# B&R Automation Studio project Panasonic_LinkaPowerCP2_A2021055 (part 6)

#### TP_Unlock.st
```iecst
(********************************************************************
 * COPYRIGHT -- Bernecker + Rainer
 ********************************************************************
 * Library: RFID
 * File: TP_Unlock.st
 * Author: houx
 * Created: March 25, 2009
*****************************************************************
;FuB: 			TP_Unlock
;*****************************************************************
Discription:
	This FuB is used to open a password-protected transponder so that all register can be edited.
	transponder key 4102 can not be used with this FuB.
	The password, protection word,and control word can only be modified after a valid TP_Unlock.
Parameter:
	Input:
		Enable(BOOL)	: The function block is only executed when enable is <> 0
	Output:
		Error(BOOL)		: Error = 0 (No Error) Error = 1(see ErrorID)
		ErrorID(UDINT)	: Number and Description in Error Table
		Busy(BOOL)		: Fub working on
		Ident(UDINT)	: Interface ID
		Done(BOOL)		: success, if TRUE
Author:	Xiaoguang Hou
		B&R Eggelsberg
;
;History:	V1.00.0 - 02 Sep 2008 : first create
				V3.00.0 - 25 Mar 2009 : update for serial interface transponder and created under AS3.0

 ********************************************************************
 * Implementation of library RFID
 ********************************************************************)

FUNCTION_BLOCK TP_Unlock

IF	(Enable	=	1)	THEN
	IF ((Done = 0) AND (Error = 0)) THEN
		Busy:=TRUE;
		IF TypeOK = FALSE THEN
			CASE StepType OF
(*	------------------------------------------------	open the interface, get the internal Ident	----------------------------------------------------*)
				OPEN:
					FrameXOpenStruct(enable := 1,device := Ident);
					status.XOPEN 			:= FrameXOpenStruct.status;
					IF (status.XOPEN = 0) THEN
						StepType            := WRITE ;
					ELSE
						StepType            := OPEN ;
						Error               := TRUE;
						ErrorID             := status.XOPEN;
						Busy                := 0;
					END_IF
				WRITE:
				memset(ADR(WriteData),0,SIZEOF(WriteData));
				strcpy(ADR(WriteData),ADR('tag,0,0,#crc$R$L'));
				FrameGetBufferStruct(enable:= 1, ident:= FrameXOpenStruct.ident);
				sendbuffer				:= FrameGetBufferStruct.buffer;
				sendbufferlength		:= FrameGetBufferStruct.buflng;
				status.GetBuffer		:= FrameGetBufferStruct.status;
				IF	(status.GetBuffer = 0)	THEN
					memcpy(sendbuffer,ADR(WriteData),sendbufferlength);
					FrameWriteStruct(enable := 1, ident := FrameXOpenStruct.ident, buffer := sendbuffer,buflng :=strlen(ADR(WriteData)));
					status.WRITE 				:=	FrameWriteStruct.status;
					StepType              		:=	READ;
				    IF (status.WRITE <> 0) THEN
						FrameReleaseOutputBufferStruct(enable:=1,ident:=FrameXOpenStruct.ident,buffer:=sendbuffer,buflng:=strlen(ADR(WriteData)));
						status.RoBuffer			:= FrameReleaseOutputBufferStruct.status;
						IF	(status.RoBuffer <> 0)	THEN
							ErrorID   	:= status.RoBuffer;
						END_IF
						FrameReleaseOutputBufferStruct.enable := 0;
						FrameWriteStruct.enable 	:=	0;
						FrameGetBufferStruct.enable	:=	0;
					END_IF
				ELSE
					ErrorID 	:= status.GetBuffer;
					Error   	:= 1;
					Busy    	:= 0;
					StepType	:= OPEN;
					TypeOK		:= FALSE;
					FrameGetBufferStruct.enable	:= 0;
				END_IF

				READ:
					FrameReadStruct(enable:=1,ident:=FrameXOpenStruct.ident);
					ReadBuffer       	:=	FrameReadStruct.buffer;
					ReadBufferLength	:=	FrameReadStruct.buflng;
					status.READ      	:=	FrameReadStruct.status;
					IF  (status.READ = 0) THEN
						memset(ADR(ReadData),0,SIZEOF(ReadData));
						memcpy(ADR(ReadData),ReadBuffer,ReadBufferLength);                   (* copy read data into read buffer *)
						FrameReadStruct.enable	:= 0;
				        FrameReleaseBufferStruct(enable:=1, ident:=FrameXOpenStruct.ident, buffer:=ReadBuffer,buflng:=ReadBufferLength);        (* release read buffer *)
				        status.ReleaseBuffer	:=FrameReleaseBufferStruct.status;
				        IF (status.ReleaseBuffer=0) THEN
					        FrameReleaseBufferStruct.enable:=0;
							AN[0]	:= ReadData[0];
							AN[1]	:= ReadData[1];
							AN[2]	:= ReadData[2];
							IF (memcmp(ADR(AN),ADR('ack'),3) = 0) THEN
								IF (memcmp(ADR(ReadData),ADR('ack,0,4150'),10) = 0) THEN
									StepType	:=	OPEN;
									TypeOK		:=	TRUE;
								ELSE
									StepType	:= 	OPEN;
									ErrorID		:=	rfidError_unlock_wrongType;          (*  hier ein Error difinieren soll  *)
									Error   	:=	1;
									Busy    	:=	0;
									TypeOK		:=	FALSE;
								END_IF
							ELSE
								StepType	:= 	OPEN;
								ErrorID		:=	rfidError_unlock_failed;          (*  hier ein Error difinieren soll  *)
								Error   	:=	1;
								Busy    	:=	0;
								TypeOK		:=	FALSE;
							END_IF
						ELSE
							StepType	:=	OPEN;
							Error     	:=	1;
							ErrorID   	:=	status.ReleaseBuffer;
							Busy      	:=	0;
							TypeOK		:=	FALSE;
						END_IF
					ELSE
						memset(ADR(ReadData),0,SIZEOF(ReadData));
					END_IF
			END_CASE
		END_IF
		IF	(TypeOK	= TRUE)	THEN
			string1	:=	'li,0,';
			string2	:=	',#crc$R$L';
			CMD		:=	strcat(ADR(string1),Data);
			CMD		:=	strcat(ADR(string1),ADR(string2));
			memset(ADR(WriteData),0,SIZEOF(WriteData));
			strcpy(ADR(WriteData),ADR(string1));
			CASE StepWrite OF
				OPEN:
					FrameXOpenStruct(enable := 1,device := Ident);
					status.XOPEN 			:= FrameXOpenStruct.status;
					IF (status.XOPEN = 0) THEN
						StepWrite            := WRITE ;
					ELSE
						StepWrite            := OPEN ;
						Error               := TRUE;
						ErrorID             := status.XOPEN;
						Busy                := 0;
					END_IF
				WRITE:
					FrameGetBufferStruct(enable:= 1, ident:= FrameXOpenStruct.ident);
					sendbuffer					:= FrameGetBufferStruct.buffer;
					sendbufferlength		:= FrameGetBufferStruct.buflng;
					status.GetBuffer		:= FrameGetBufferStruct.status;
					IF	(status.GetBuffer = 0)	THEN
						memcpy(sendbuffer,ADR(WriteData),sendbufferlength);
						FrameWriteStruct(enable := 1, ident := FrameXOpenStruct.ident, buffer := sendbuffer,buflng := strlen(ADR(WriteData)));
						status.WRITE 				:=	FrameWriteStruct.status;
					    IF (status.WRITE = FALSE) THEN
					    	StepWrite              		:=	READ;
							FrameWriteStruct.enable 	:=	0;
							FrameGetBufferStruct.enable	:=	0;
						ELSE
							ErrorID 				:= status.WRITE;
							Error   				:= 1;
							Busy    				:= 0;
							StepWrite				:= OPEN;
							TypeOK					:= FALSE;
							FrameWriteStruct.enable := 0;
							FrameGetBufferStruct.enable	:= 0;
							FrameReleaseOutputBufferStruct(enable:=1,ident:=FrameXOpenStruct.ident,buffer:=sendbuffer,buflng:= sendbufferlength);
							status.RoBuffer			:= FrameReleaseOutputBufferStruct.status;
							IF	(status.RoBuffer <> 0)	THEN
								StepWrite 	:= OPEN;
								Error     	:= TRUE;
								ErrorID   	:= status.RoBuffer;
								Busy      	:= 0;
								TypeOK		:= FALSE;
								FrameReleaseOutputBufferStruct.enable := 0;
							END_IF
						END_IF
					ELSE
						ErrorID 	:= status.GetBuffer;
						Error   	:= 1;
						Busy    	:= 0;
						StepWrite	:= OPEN;
						TypeOK		:= FALSE;
						FrameGetBufferStruct.enable	:= 0;
					END_IF
			    READ:
				    FrameReadStruct(enable := 1,ident:=FrameXOpenStruct.ident);
					ReadBuffer			:=	FrameReadStruct.buffer;
					ReadBufferLength	:=	FrameReadStruct.buflng;
					status.READ			:=	FrameReadStruct.status;
					IF  (status.READ = 0)  THEN
						memset(ADR(ReadData),0,SIZEOF(ReadData));
						memcpy(ADR(ReadData),ReadBuffer,ReadBufferLength);
						FrameReadStruct.enable := 0;
				        FrameReleaseBufferStruct(enable:=1, ident:=FrameXOpenStruct.ident, buffer:=ReadBuffer,buflng:=ReadBufferLength);
				        status.ReleaseBuffer	:=	FrameReleaseBufferStruct.status;
				        IF status.ReleaseBuffer=0 THEN
							FrameReleaseBufferStruct.enable:=0;
							AN[0]	:= ReadData[0];
							AN[1]	:= ReadData[1];
							AN[2]	:= ReadData[2];
							IF (memcmp(ADR(AN),ADR('ack'),3)) = 0 THEN
								StepWrite		:=	WRITE;
							 	Busy			:=	0;
							 	Done			:=	1;
								TypeOK			:=	FALSE;
							ELSIF	(memcmp(ADR(AN),ADR('nak'),3)) = 0 THEN
								ERROR[0]	:=	ReadData[6];
								ERROR[1]	:=	ReadData[7];
								ERROR[2]	:=	ReadData[8];
								Error		:=	1;
								ErrorID		:=	atoi(ADR(ERROR)) ;
								Busy		:=	0;
								TypeOK		:=	FALSE;
								StepWrite	:=	WRITE;
							ELSE
								Error			:=	1;
								ErrorID			:=	rfidError_unlock_failed ;(* unknow answer *)
								Busy			:=	0;
								TypeOK			:=	FALSE;
								StepWrite		:=	WRITE;
							END_IF
						ELSE
							Error			:=	1;
							ErrorID			:=	status.ReleaseBuffer ;
							Busy			:=	0;
							TypeOK			:=	FALSE;
							StepWrite		:=	WRITE;
					    END_IF
					ELSE
						memset(ADR(ReadData),0,SIZEOF(ReadData));
					END_IF
			END_CASE
		END_IF
	END_IF
ELSE
	Busy	:=	0;
	Error	:=	0;
	ErrorID	:=	0;
	Done	:=	0;
END_IF
END_FUNCTION_BLOCK
```

#### TP_Lock.st
```iecst
(********************************************************************
 * COPYRIGHT -- Bernecker + Rainer
 ********************************************************************
 * Library: RFID
 * File: TP_Lock.st
 * Author: houx
 * Created: March 25, 2009
 *****************************************************************
;FuB: 			TP_Lock
;*****************************************************************
Discription:
	If a password-protected transponder was opened with the TP_Unlock, it can be locked again with this FuB
	From this point on, password-protected areas can no longer be edited.
	if the transponder is removed from the reading range of the transponder reader, then it is locked automatically.
Parameter:
	Input:
		Enable(BOOL)	: The function block is only executed when enable is <> 0
	Output:
		Error(BOOL)		: Error = 0 (No Error) Error = 1(see ErrorID)
		ErrorID(UDINT)	: Number and Description in Error Table
		Busy(BOOL)		: Fub working on
		Ident(UDINT)	: Interface ID
		Done(BOOL)		: success, if TRUE
;Author:	Xiaoguang Hou
;			B&R Eggelsberg
;
;History:	V1.00.0 - 02 Sep 2008 : first create
				V3.00.0 - 25 Mar 2009 : update for serial interface transponder and created under AS3.0
;
;******************************************************************

 ********************************************************************
 * Implementation of library RFID
 ********************************************************************)
(*TODO: Add your comment here*)
FUNCTION_BLOCK TP_Lock

IF Enable = TRUE THEN
	IF ((Done = 0) AND (Error = 0)) THEN
		Busy:=TRUE;
		IF TypeOK = FALSE THEN
			CASE StepType OF
(*	------------------------------------------------	open the interface, get the internal Ident	----------------------------------------------------*)
				OPEN:
					FrameXOpenStruct(enable := 1,device := Ident);
					status.XOPEN 			:= FrameXOpenStruct.status;
					IF (status.XOPEN = 0) THEN
						StepType            := WRITE ;
					ELSE
						StepType            := OPEN ;
						Error               := TRUE;
						ErrorID             := status.XOPEN;
						Busy                := 0;
					END_IF
				WRITE:
					memset(ADR(WriteData),0,SIZEOF(WriteData));
					strcpy(ADR(WriteData),ADR('tag,0,0,#crc$R$L'));
					FrameGetBufferStruct(enable:= 1, ident:= FrameXOpenStruct.ident);
					sendbuffer				:= FrameGetBufferStruct.buffer;
					sendbufferlength		:= FrameGetBufferStruct.buflng;
					status.GetBuffer		:= FrameGetBufferStruct.status;
					IF	(status.GetBuffer = 0)	THEN
						memcpy(sendbuffer,ADR(WriteData),sendbufferlength);
						FrameWriteStruct(enable := 1, ident := FrameXOpenStruct.ident, buffer := sendbuffer,buflng := strlen(ADR(WriteData)));
						status.WRITE 				:=	FrameWriteStruct.status;
					    StepType              		:=	READ;
					    IF (status.WRITE <> 0) THEN
							FrameReleaseOutputBufferStruct(enable:=1,ident:=FrameXOpenStruct.ident,buffer:=sendbuffer,buflng:= strlen(ADR(WriteData)));
							status.RoBuffer			:= FrameReleaseOutputBufferStruct.status;
							IF	(status.RoBuffer <> 0)	THEN
								ErrorID   	:= status.RoBuffer;
							END_IF
						END_IF
						FrameWriteStruct.enable := 0;
						FrameGetBufferStruct.enable	:= 0;
						FrameReleaseOutputBufferStruct.enable := 0;
					ELSE
						ErrorID 	:= status.GetBuffer;
						Error   	:= 1;
						Busy    	:= 0;
						StepType	:= OPEN;
						TypeOK		:= FALSE;
						FrameGetBufferStruct.enable	:= 0;
					END_IF
				READ:
					FrameReadStruct(enable:=1,ident:=FrameXOpenStruct.ident);
					ReadBuffer       	:=	FrameReadStruct.buffer;
					ReadBufferLength	:=	FrameReadStruct.buflng;
					status.READ      	:=	FrameReadStruct.status;
					IF  (status.READ = 0) THEN
						memset(ADR(ReadData),0,SIZEOF(ReadData));
						memcpy(ADR(ReadData),ReadBuffer,ReadBufferLength);                   (* copy read data into read buffer *)
						FrameReadStruct.enable	:= 0;
				        FrameReleaseBufferStruct(enable:=1, ident:=FrameXOpenStruct.ident, buffer:=ReadBuffer,buflng:=ReadBufferLength);        (* release read buffer *)
				        status.ReleaseBuffer	:=FrameReleaseBufferStruct.status;
				        IF (status.ReleaseBuffer=0) THEN
					        FrameReleaseBufferStruct.enable:=0;
							AN[0]	:= ReadData[0];
							AN[1]	:= ReadData[1];
							AN[2]	:= ReadData[2];
							IF (memcmp(ADR(AN),ADR('ack'),3) = 0) THEN
								IF (memcmp(ADR(ReadData),ADR('ack,0,4150,#02d0$R$L'),SIZEOF('ack,0,4150,#02d0$R$L')) = 0) THEN
									StepType	:=	OPEN;
									TypeOK		:=	TRUE;
									StepLOCK	:=	WRITE;
								ELSE
									StepType	:= 	OPEN;
									ErrorID		:=	rfidError_lock_wrongType;          (*  hier ein Error difinieren soll  *)
									Error   	:=	1;
									Busy    	:=	0;
									TypeOK		:=	FALSE;
								END_IF
							ELSE
								StepType	:= 	OPEN;
								ErrorID		:=	rfidError_lock_failed;          (*  hier ein Error difinieren soll  *)
								Error   	:=	1;
								Busy    	:=	0;
								TypeOK		:=	FALSE;
							END_IF
						ELSE
							StepType	:=	OPEN;
							Error     	:=	1;
							ErrorID   	:=	status.ReleaseBuffer;
							Busy      	:=	0;
							TypeOK		:=	FALSE;
						END_IF
					ELSE
						memset(ADR(ReadData),0,SIZEOF(ReadData));
					END_IF
			END_CASE
		END_IF
		IF TypeOK = TRUE THEN
			CASE StepLOCK OF
				WRITE:
					memset(ADR(WriteData),0,SIZEOF(WriteData));
					strcpy(ADR(WriteData),ADR('re,0,#crc$R$L'));
					FrameGetBufferStruct(enable:= 1, ident:= FrameXOpenStruct.ident);
					sendbuffer				:= FrameGetBufferStruct.buffer;
					sendbufferlength		:= FrameGetBufferStruct.buflng;
					status.GetBuffer		:= FrameGetBufferStruct.status;
					IF	(status.GetBuffer = 0)	THEN
						memcpy(sendbuffer,ADR(WriteData),sendbufferlength);
						FrameWriteStruct(enable := 1, ident := FrameXOpenStruct.ident, buffer := sendbuffer,buflng := strlen(ADR(WriteData)));
						status.WRITE 				:=	FrameWriteStruct.status;
					   	StepLOCK              		:=	READ;
					    IF (status.WRITE <> 0) THEN
							FrameReleaseOutputBufferStruct(enable:=1,ident:=FrameXOpenStruct.ident,buffer:=sendbuffer,buflng:= sendbufferlength);
							status.RoBuffer			:= FrameReleaseOutputBufferStruct.status;
							IF	(status.RoBuffer <> 0)	THEN
								ErrorID   	:= status.RoBuffer;
							END_IF
						END_IF
						FrameWriteStruct.enable := 0;
						FrameGetBufferStruct.enable	:= 0;
						FrameReleaseOutputBufferStruct.enable := 0;
					ELSE
						ErrorID 	:= status.GetBuffer;
						Error   	:= 1;
						Busy    	:= 0;
						StepLOCK	:= WRITE;
						TypeOK		:= FALSE;
						FrameGetBufferStruct.enable	:= 0;
					END_IF
				READ:
				    FrameReadStruct(enable := 1,ident:=FrameXOpenStruct.ident);
					ReadBuffer			:= FrameReadStruct.buffer;
					ReadBufferLength	:= FrameReadStruct.buflng;
					status.READ			:= FrameReadStruct.status;
					IF  (status.READ = 0) THEN
						memset(ADR(ReadData),0,SIZEOF(ReadData));
						memcpy(ADR(ReadData),ReadBuffer,ReadBufferLength);                   (* copy read data into read buffer *)
						FrameReadStruct.enable 	:= 0;
				        FrameReleaseBufferStruct(enable:=1, ident:=FrameXOpenStruct.ident, buffer:=ReadBuffer,buflng:=ReadBufferLength);        (* release read buffer *)
				        status.ReleaseBuffer	:= FrameReleaseBufferStruct.status;
				        IF (status.ReleaseBuffer=0) THEN
						    FrameReleaseBufferStruct.enable	:= 0;
							AN[0]	:= ReadData[0];
							AN[1]	:= ReadData[1];
							AN[2]	:= ReadData[2];
							IF (memcmp(ADR(AN),ADR('ack'),3)) = 0 THEN
								StepLOCK  := WRITE;
								Done      := 1;
								Busy      := 0;
								TypeOK	  := FALSE;
							ELSIF	(memcmp(ADR(AN),ADR('nak'),3)) = 0 THEN
								ERROR[0]	:=	ReadData[6];
								ERROR[1]	:=	ReadData[7];
								ERROR[2]	:=	ReadData[8];
								Error		:=	1;
								ErrorID		:=	atoi(ADR(ERROR)) ;
								Busy		:=	0;
								TypeOK		:=	FALSE;
								StepLOCK	:=	WRITE;
							ELSE
								StepLOCK  := WRITE;
								Error     := 1;
								ErrorID   := rfidError_lock_failed; (* unknow answer *)
								Busy      := 0;
								TypeOK	  := FALSE;
							END_IF
						ELSE
							StepLOCK  := WRITE;
							Error     := 1;
							ErrorID   := status.ReleaseBuffer;
							Busy      := 0;
							TypeOK	  := FALSE;
					    END_IF
					ELSE
						memset(ADR(ReadData),0,SIZEOF(ReadData));
					END_IF
			END_CASE
		END_IF
	END_IF
ELSE
	Busy 	:= 0;
	ErrorID := 0;
	Error 	:= 0;
	Done 	:= 0;
END_IF
END_FUNCTION_BLOCK
```

#### TP_PWProtect.st
```iecst
(********************************************************************
 * COPYRIGHT -- Bernecker + Rainer
 ********************************************************************
 * Library: RFID
 * File: TP_PWProtect.st
 * Author: houx
 * Created: March 25, 2009
 *****************************************************************
;FuB: 			TP_PWProtect
;*****************************************************************
Discription:
	This FuB is used to write the password
	before a new password can be written, a valid TP_Unlock must be done.
Parameter:
	Input:
		Enable(BOOL)	:The function block is only executed when enable is <> 0
		Data(UDINT)		:Pointer to Password. whick should be write in transponder.
	Output:
		Error(BOOL)		:Error = 0 (No Error) Error = 1(see ErrorID)
		ErrorID(UDINT)	:Number and Description in Error Table
		Busy(BOOL)		:Fub working on
		Done			:success, if TRUE
;Author:	Xiaoguang Hou
;			B&R Eggelsberg
;
;History: 	V1.00.0 - 02 Sep 2008 first create
				V3.00.0 - 25 Mar 2009  update for serial interface transponder reader and created under AS3.0
;
;******************************************************************

 ********************************************************************
 * Implementation of library RFID
 ********************************************************************)

(*TODO: Add your comment here*)
FUNCTION_BLOCK TP_PWProtect

IF	(Enable	=	1)	THEN
	IF ((Done = 0) AND (Error = 0)) THEN
		Busy:=TRUE;
		IF TypeOK = FALSE THEN
			CASE StepType OF
(*	------------------------------------------------	open the interface, get the internal Ident	----------------------------------------------------*)
				OPEN:
					FrameXOpenStruct(enable := 1,device := Ident);
					status.XOPEN 			:= FrameXOpenStruct.status;
					IF (status.XOPEN = 0) THEN
						StepType            := WRITE ;
					ELSE
						StepType            := OPEN ;
						Error               := TRUE;
						ErrorID             := status.XOPEN;
						Busy                := 0;
					END_IF
				WRITE:
					memset(ADR(WriteData),0,SIZEOF(WriteData));
					strcpy(ADR(WriteData),ADR('tag,0,0,#crc$R$L'));
					FrameGetBufferStruct(enable:= 1, ident:= FrameXOpenStruct.ident);
					sendbuffer				:= FrameGetBufferStruct.buffer;
					sendbufferlength		:= FrameGetBufferStruct.buflng;
					status.GetBuffer		:= FrameGetBufferStruct.status;
					IF	(status.GetBuffer = 0)	THEN
						memcpy(sendbuffer,ADR(WriteData),sendbufferlength);
						FrameWriteStruct(enable := 1, ident := FrameXOpenStruct.ident, buffer := sendbuffer,buflng := strlen(ADR(WriteData)));
						status.WRITE 				:=	FrameWriteStruct.status;
					    StepType              		:=	READ;
					    IF (status.WRITE <> 0) THEN
							FrameReleaseOutputBufferStruct(enable:=1,ident:=FrameXOpenStruct.ident,buffer:=sendbuffer,buflng:= strlen(ADR(WriteData)));
							status.RoBuffer			:= FrameReleaseOutputBufferStruct.status;
							IF	(status.RoBuffer <> 0)	THEN
								ErrorID	:=	status.RoBuffer;
							END_IF
						END_IF
						FrameWriteStruct.enable := 0;
						FrameGetBufferStruct.enable	:= 0;
						FrameReleaseOutputBufferStruct.enable := 0;
					ELSE
						ErrorID 	:= status.GetBuffer;
						Error   	:= 1;
						Busy    	:= 0;
						StepType	:= OPEN;
						TypeOK		:= FALSE;
						FrameGetBufferStruct.enable	:= 0;
					END_IF

				READ:
					FrameReadStruct(enable:=1,ident:=FrameXOpenStruct.ident);
					ReadBuffer       	:=	FrameReadStruct.buffer;
					ReadBufferLength	:=	FrameReadStruct.buflng;
					status.READ      	:=	FrameReadStruct.status;
					IF  (status.READ = 0) THEN
						memset(ADR(ReadData),0,SIZEOF(ReadData));
						memcpy(ADR(ReadData),ReadBuffer,ReadBufferLength);                   (* copy read data into read buffer *)
						FrameReadStruct.enable	:= 0;
				        FrameReleaseBufferStruct(enable:=1, ident:=FrameXOpenStruct.ident, buffer:=ReadBuffer,buflng:=ReadBufferLength);        (* release read buffer *)
				        status.ReleaseBuffer	:=FrameReleaseBufferStruct.status;
				        IF (status.ReleaseBuffer=0) THEN
					        FrameReleaseBufferStruct.enable:=0;
							IF (memcmp(ADR(ReadData),ADR('ack,0,4150,#02d0$R$L'),SIZEOF('ack,0,4150,#02d0$R$L')) = 0) THEN
								StepType	:=	OPEN;
								TypeOK		:=	TRUE;
								StepWrite	:=	WRITE;
							ELSE
								StepType	:= 	OPEN;
								ErrorID		:=	rfidError_password_wrongType;         (*   hier ein Error difinieren soll  *)
								Error   	:=	1;
								Busy    	:=	0;
								TypeOK		:=	FALSE;
							END_IF
						ELSE
							StepType	:=	OPEN;
							Error     	:=	1;
							ErrorID   	:=	status.ReleaseBuffer;
							Busy      	:=	0;
							TypeOK		:=	FALSE;
						END_IF
					ELSE
						memset(ADR(ReadData),0,SIZEOF(ReadData));
					END_IF
			END_CASE
		END_IF
		IF	(TypeOK	= TRUE)	THEN
			string1	:=	'wp,0,';
			string2	:=	',#crc$R$L';
			CMD		:=	strcat(ADR(string1),Data);
			CMD		:=	strcat(ADR(string1),ADR(string2));
			memset(ADR(WriteData),0,SIZEOF(WriteData));
			memcpy(ADR(WriteData),ADR(string1),SIZEOF(string1));
			CASE StepWrite OF
				WRITE:
					FrameGetBufferStruct(enable:= 1, ident:= FrameXOpenStruct.ident);
					sendbuffer				:= FrameGetBufferStruct.buffer;
					sendbufferlength		:= FrameGetBufferStruct.buflng;
					status.GetBuffer		:= FrameGetBufferStruct.status;
					IF	(status.GetBuffer = 0)	THEN
						memcpy(sendbuffer,ADR(WriteData),sendbufferlength);
						FrameWriteStruct(enable := 1, ident := FrameXOpenStruct.ident, buffer := sendbuffer,buflng := strlen(ADR(WriteData)));
						status.WRITE 				:=	FrameWriteStruct.status;
					    StepWrite              		:=	READ;
					    IF (status.WRITE <> 0) THEN
							FrameReleaseOutputBufferStruct(enable:=1,ident:=FrameXOpenStruct.ident,buffer:=sendbuffer,buflng:=strlen(ADR(WriteData)) );
							status.RoBuffer			:= FrameReleaseOutputBufferStruct.status;
							IF	(status.RoBuffer <> 0)	THEN
								ErrorID	:=	status.RoBuffer;
							END_IF
						END_IF
						FrameWriteStruct.enable := 0;
						FrameGetBufferStruct.enable	:= 0;
						FrameReleaseOutputBufferStruct.enable := 0;
					ELSE
						ErrorID 	:= status.GetBuffer;
						Error   	:= 1;
						Busy    	:= 0;
						StepWrite	:= WRITE;
						TypeOK		:= FALSE;
						FrameGetBufferStruct.enable	:= 0;
					END_IF

			    READ:
				    FrameReadStruct(enable := 1,ident:=FrameXOpenStruct.ident);
					ReadBuffer			:=	FrameReadStruct.buffer;
					ReadBufferLength	:=	FrameReadStruct.buflng;
					status.READ			:=	FrameReadStruct.status;
					IF  (status.READ = 0)  THEN
						memset(ADR(ReadData),0,SIZEOF(ReadData));
						memcpy(ADR(ReadData),ReadBuffer,ReadBufferLength);
						FrameReadStruct.enable := 0;
				        FrameReleaseBufferStruct(enable:=1, ident:=FrameXOpenStruct.ident, buffer:=ReadBuffer,buflng:=ReadBufferLength);
				        status.ReleaseBuffer	:=	FrameReleaseBufferStruct.status;
				        IF status.ReleaseBuffer=0 THEN
							FrameReleaseBufferStruct.enable:=0;
							memset(ADR(AN),0,SIZEOF(AN));
							AN[0]	:= ReadData[0];
							AN[1]	:= ReadData[1];
							AN[2]	:= ReadData[2];
							IF (memcmp(ADR(AN),ADR('ack'),3)) = 0 THEN
								StepWrite		:=	WRITE;
							 	Busy			:=	0;
							 	Done			:=	1;
								TypeOK			:=	FALSE;
							ELSIF	(memcmp(ADR(AN),ADR('nak'),3)) = 0 THEN
								ERROR[0]	:=	ReadData[6];
								ERROR[1]	:=	ReadData[7];
								ERROR[2]	:=	ReadData[8];
								Error			:=	1;
								ErrorID			:=	atoi(ADR(ERROR)) ;
								Busy			:=	0;
								TypeOK			:=	FALSE;
								StepWrite		:=	WRITE;
							ELSE
								Error			:=	1;
								ErrorID			:=	rfidError_password_failed ;
								Busy			:=	0;
								TypeOK			:=	FALSE;
								StepWrite		:=	WRITE;
							END_IF
						ELSE
							Error			:=	1;
							ErrorID			:=	status.ReleaseBuffer ;
							Busy			:=	0;
							TypeOK			:=	FALSE;
							StepWrite		:=	WRITE;
					    END_IF
					ELSE
						memset(ADR(ReadData),0,SIZEOF(ReadData));
					END_IF
			END_CASE
		END_IF
	END_IF
ELSE
	Busy	:=	0;
	Error	:=	0;
	ErrorID	:=	0;
	Done	:=	0;
END_IF
END_FUNCTION_BLOCK
```

#### TP_OnOff.st
```iecst
(********************************************************************
 * COPYRIGHT -- Bernecker + Rainer
 ********************************************************************
 * Library: RFID
 * File: TP_OnOff.st
 * Author: houx
 * Created: March 25, 2009
 *****************************************************************
;FuB: 			TP_OnOff
;*****************************************************************
Discription:
	This FuB turn the 125 kHz carrier frequency of the Transponder reader/writer On/Off.
	This Fub can work without any Transponder in the range of Reader.
	Standard Configuration is frequency on.
	Be aware that no Transponder key can be read if frequency is turned off.
Parameter:
	Input:
		Enable(BOOL)	:	The function block is only executed when enable is <> 0
		Ident(UDINT)	:	Interface Ident from TP_Init.
   		Mode(BOOL)		:	frequency On:Mode=TRUE, frequency Off: Mode:=FALSE;
	Output:
		Error(BOOL)		:	Error = 0 (No Error) Error = 1(see ErrorID)
		ErrorID(UDINT)	:	Number and Description in Error Table
		Busy(BOOL)		:	if TRUE , Fub working on.
		Done(BOOL) 		:	if TRUE, success
Author:	Xiaoguang Hou
		B&R Eggelsberg

History: 	V1.00.0 - 02 Sep 2008 first create
				V3.00.0 - 25 Mar 2009  update for serial interface transponder reader and created under AS3.0

;******************************************************************

 ********************************************************************
 * Implementation of library RFID
 ********************************************************************)

(*TODO: Add your comment here*)
FUNCTION_BLOCK TP_OnOff

(*------------------------------------	Start	--------------------------------*)
IF Enable=1 THEN
	IF ((Done = 0) AND (Error = 0)) THEN
		Busy:=TRUE;
		CASE StepOnOff OF
(*	------------------------------------------------	open the interface, get the internal Ident	----------------------------------------------------*)
			OPEN:
				FrameXOpenStruct(enable := TRUE,device := Ident);
				status.XOPEN 			:= FrameXOpenStruct.status;
				IF (status.XOPEN = 0) THEN
					StepOnOff               := WRITE ;
					FrameXOpenStruct.enable:=FALSE;
				ELSE
					StepOnOff               := OPEN ;
					Error                   := TRUE;
					ErrorID                 := status.XOPEN;
					Busy                    := FALSE;
				END_IF

			WRITE:						(*------	write RF Command to	Reader	---------*)
				IF (Mode = TRUE) THEN
					memset(ADR(WriteData),0,SIZEOF(WriteData));
					strcpy(ADR(WriteData),ADR('rf,0,1,#crc$R$L'));
				ELSIF	(Mode = FALSE)	THEN
					memset(ADR(WriteData),0,SIZEOF(WriteData));
					strcpy(ADR(WriteData),ADR('rf,0,0,#crc$R$L'));
				END_IF
				(*------	get sendbuffer	---------*)
				FrameGetBufferStruct(enable:= TRUE, ident:= FrameXOpenStruct.ident);
				sendbuffer				:= FrameGetBufferStruct.buffer;
				sendbufferlength		:= FrameGetBufferStruct.buflng;
				status.GetBuffer		:= FrameGetBufferStruct.status;
				IF	(status.GetBuffer = 0)	THEN							 (*------	no error	---------*)
					memcpy(sendbuffer,ADR(WriteData),sendbufferlength);
					FrameWriteStruct(enable := TRUE, ident := FrameXOpenStruct.ident, buffer := sendbuffer,buflng :=strlen(ADR(WriteData)) );
					status.WRITE 				:=	FrameWriteStruct.status;
			        IF (status.WRITE <> 0) THEN
						FrameReleaseOutputBufferStruct(enable:=TRUE,ident:=FrameXOpenStruct.ident,buffer:=sendbuffer,buflng:= strlen(ADR(WriteData)));
						status.RoBuffer			:= FrameReleaseOutputBufferStruct.status;
						IF	(status.RoBuffer <> 0)	THEN
							ErrorID	:=	status.RoBuffer;
						END_IF
					ELSE
			        	StepOnOff              		:=	READ;
						FrameWriteStruct.enable := FALSE;
						FrameGetBufferStruct.enable	:= FALSE;
						FrameReleaseOutputBufferStruct.enable := FALSE;
					END_IF
				(*------	if get sendbuffer error	---------*)
				ELSE
					ErrorID 	:= status.GetBuffer;
					Error   	:= TRUE;
					Busy    	:= FALSE;
					StepOnOff	:= OPEN;
					FrameGetBufferStruct.enable	:= FALSE;
				END_IF

	    	READ:						(*	read out the feedback	*)
			    FrameReadStruct(enable := 1,ident:=FrameXOpenStruct.ident);
				ReadBuffer				:=FrameReadStruct.buffer;
				ReadBufferLength		:=FrameReadStruct.buflng;
				status.READ				:=FrameReadStruct.status;
				IF  (status.READ = 0) THEN
					memset(ADR(ReadData),0,SIZEOF(ReadData));
					memcpy(ADR(ReadData),ReadBuffer,ReadBufferLength);	(*	copy the answer	out in ReadData	*)
					FrameReadStruct.enable := 0;
			        FrameReleaseBufferStruct(enable:=1, ident:=FrameXOpenStruct.ident, buffer:=ReadBuffer,buflng:=ReadBufferLength);	(*	release the buffer	*)
			        status.ReleaseBuffer   := FrameReleaseBufferStruct.status;
			        IF (status.ReleaseBuffer=0) THEN
			        	FrameReleaseBufferStruct.enable	:= 0;
			        	AN[0]	:= ReadData[0];
						AN[1]	:= ReadData[1];
						AN[2]	:= ReadData[2];
						IF (memcmp(ADR(AN),ADR('ack'),3) = 0) THEN				(*--- positiv answer ----*)
							StepOnOff   := CLOSE;
						ELSE
							StepOnOff   := OPEN;								(*	negativ answer or unknow answer	*)
							Error     	:= 1;
							ErrorID   	:= rfidError_rf_failed;
							Busy      	:= 0;
						END_IF
					ELSE														(*	if buffer release error	*)
							StepOnOff   := OPEN;
							Error     	:= 1;
							ErrorID   	:= status.ReleaseBuffer;
							Busy     	:= 0;
			        END_IF
				ELSE
					memset(ADR(ReadData),0,SIZEOF(ReadData));
				END_IF
			CLOSE:
				FRM_close_0(enable :=1 , ident :=FrameXOpenStruct.ident);
				IF FRM_close_0.status=FALSE THEN
					Done      	:= 1;
					Busy      	:= 0;
					StepOnOff:=OPEN;
				END_IF
		END_CASE
	END_IF
ELSE                                          (*------- if enable = False ,then all output variable back to zero -------*)
	Error:=0;
	ErrorID:=0;
	Busy:=0;
	Done:=0;
END_IF
END_FUNCTION_BLOCK
```

#### TP_Crc.st
```iecst
(********************************************************************
 * COPYRIGHT -- Bernecker + Rainer
 ********************************************************************
 * Library: RFID
 * File: TP_Crc.st
 * Author: houx
 * Created: March 25, 2009
*****************************************************************
;FuB: 			TP_CRC
;*****************************************************************
Discription:
	This FuB can specify whether the transponder reader should check the checksum wenn a command string is received.
	This Fub can work without any Transponder in the range of Reader.
Parameter:
	Input: 	Enable(BOOL)	: The function block is only executed when enable is <> 0.
			Ident(UDINT)	: Interface Ident.
			Mode(BOOL)		: checksum On:Mode=TRUE, checksum Off: Mode:=FALSE;
	Output: Error(BOOL)		: Error = 0 (No Error) Error = 1(see ErrorID).
			ErrorID(UDINT)	: Number and description in error table.
			Busy(BOOL)		: FuB is working on.
			Done(BOOL)		: if TRUE, success.
Author:	Xiaoguang Hou
		B&R Eggelsberg

History: 	V1.00.0 - 02 Sep 2008 first create
				V3.00.0 - 25 Mar 2009  update for serial interface transponder readerand created under AS3.0
;
;******************************************************************

 ********************************************************************
 * Implementation of library RFID
 ********************************************************************)

(*TODO: Add your comment here*)
FUNCTION_BLOCK TP_Crc

IF Enable=1 THEN
	IF ((Done = 0) AND (Error = 0)) THEN
		Busy:=TRUE;
		CASE StepCRC OF
(*	------------------------------------------------	open the interface, get the internal Ident	----------------------------------------------------*)
			OPEN:
				FrameXOpenStruct(enable := 1,device := Ident);
				status.XOPEN 			:= FrameXOpenStruct.status;
				IF (status.XOPEN = 0) THEN
					StepCRC             := WRITE ;
					FrameXOpenStruct.enable:=FALSE;
				ELSE
					StepCRC             := OPEN ;
					Error               := TRUE;
					ErrorID             := status.XOPEN;
					Busy                := 0;
				END_IF
			WRITE:
				IF 	(Mode = TRUE) THEN
					memset(ADR(WriteData),0,SIZEOF(WriteData));
					strcpy(ADR(WriteData),ADR('cc,0,1,#01ce$R$L'));
				ELSIF (Mode = FALSE) THEN
					memset(ADR(WriteData),0,SIZEOF(WriteData));
					strcpy(ADR(WriteData),ADR('cc,0,0,#01cd$R$L'));
				END_IF
				FrameGetBufferStruct(enable:= 1, ident:= FrameXOpenStruct.ident);
				sendbuffer				:= FrameGetBufferStruct.buffer;
				sendbufferlength		:= FrameGetBufferStruct.buflng;
				status.GetBuffer		:= FrameGetBufferStruct.status;
				IF	(status.GetBuffer = 0)	THEN
					memcpy(sendbuffer,ADR(WriteData),sendbufferlength);
					FrameWriteStruct(enable := 1, ident := FrameXOpenStruct.ident, buffer := sendbuffer, buflng := strlen(ADR(WriteData)));
					status.WRITE 				:=	FrameWriteStruct.status;

			    	IF (status.WRITE <> 0) THEN
						FrameReleaseOutputBufferStruct(enable:=1,ident:=FrameXOpenStruct.ident,buffer:=sendbuffer,buflng:= strlen(ADR(WriteData)));
						status.RoBuffer			:= FrameReleaseOutputBufferStruct.status;
						IF	(status.RoBuffer <> 0)	THEN
							ErrorID:=status.RoBuffer;
						END_IF
					ELSE
			   			FrameWriteStruct.enable := 0;
						FrameGetBufferStruct.enable	:= 0;
						FrameReleaseOutputBufferStruct.enable := 0;
						StepCRC					:= READ;
					END_IF
				ELSE
					ErrorID 	:= status.GetBuffer;
					Error   	:= 1;
					Busy    	:= 0;
					StepCRC		:= OPEN;
					FrameGetBufferStruct.enable	:= 0;
				END_IF

		    READ:
			    FrameReadStruct(enable := 1,ident:=FrameXOpenStruct.ident);
				ReadBuffer			:= FrameReadStruct.buffer;
				ReadBufferLength	:= FrameReadStruct.buflng;
				status.READ			:= FrameReadStruct.status;
				IF  (status.READ = 0) THEN
					memset(ADR(ReadData),0,SIZEOF(ReadData));
					memcpy(ADR(ReadData),ReadBuffer,ReadBufferLength);                   (* copy read data into read buffer *)
					FrameReadStruct.enable 	:= 0;
			        FrameReleaseBufferStruct(enable:=1, ident:=FrameXOpenStruct.ident, buffer:=ReadBuffer,buflng:=ReadBufferLength);        (* release read buffer *)
			        status.ReleaseBuffer	:= FrameReleaseBufferStruct.status;
			        IF (status.ReleaseBuffer=0) THEN
				        FrameReleaseBufferStruct.enable	:=0;
		        		AN[0]	:= ReadData[0];
						AN[1]	:= ReadData[1];
						AN[2]	:= ReadData[2];
						IF (memcmp(ADR(AN),ADR('ack'),3) = 0) THEN
							StepCRC   := CLOSE;
						ELSE
							StepCRC   := OPEN;
							Error     := 1;
							ErrorID   := rfidError_crc_failed; (*	negativ answer *)
							Busy      := 0;
						END_IF
					ELSE
							StepCRC   := OPEN;
							Error     := 1;
							ErrorID   := status.ReleaseBuffer;
							Busy      := 0;
			        END_IF
				ELSE
					memset(ADR(ReadData),0,SIZEOF(ReadData));
				END_IF
			CLOSE:
				FRM_close_0(enable :=1 , ident :=FrameXOpenStruct.ident);
				IF FRM_close_0.status=FALSE  THEN
					Done      := 1;
					Busy      := 0;
					StepCRC   := OPEN;
				END_IF
		END_CASE
	END_IF
ELSE
	Error   := 0;
	ErrorID := 0;
	Busy    := 0;
	Done    := 0;
END_IF

END_FUNCTION_BLOCK
```

#### TP_Write.st
```iecst
(********************************************************************
 * COPYRIGHT -- Bernecker + Rainer
 ********************************************************************
 * Library: RFID
 * File: TP_Write.st
 * Author: houx
 * Created: March 25, 2009
 ****************************************************************
;FuB: 			TP_Write
;*****************************************************************
Discription:
	This FuB is used to write the registers of the transponder.
	for this to work, the transponder must not be password-protected or a valid TP_unlock must be carried out beforehand.
	Be aware that Register 1 and 2 of TP 4150 are used for the control and protectionwords.
	Only modify these registers,if you are familiar with their Function. In addition, avalid login is needed.
Parameter:
	Input:
		Enable(BOOL)	: The function block is only executed when enable is <> 0
		RegNr(USINT)	: Number of the register, which should be write in
		Data(UDINT)		: pointer to input Data
	Output:
		Error(BOOL)		: Error = 0 (No Error) Error = 1(see ErrorID)
		ErrorID(UDINT)	: Number and Description in Error Table
		Busy(BOOL)		: Fub working on
		Ident(UDINT)	: Interface ID
		Done(BOOL)		:success, if TRUE
Author:	Xiaoguang Hou
		B&R Eggelsberg
;
History: 	V1.00.0 - 02 Sep 2008 first create
				V3.00.0 - 25 Mar 2009  update for serial interface transponder reader and created under AS3.0
;
 ********************************************************************
 * Implementation of library RFID
 ********************************************************************)

(*TODO: Add your comment here*)
FUNCTION_BLOCK TP_Write

IF (Enable = 1) THEN
	IF ((Done = 0) AND (Error = 0)) THEN
		Busy:=TRUE;
		IF TypeOK = FALSE THEN
			CASE StepType OF
(*	------------------------------------------------	open the interface, get the internal Ident	----------------------------------------------------*)
				OPEN:
					FrameXOpenStruct(enable := 1,device := Ident);
					status.XOPEN 			:= FrameXOpenStruct.status;
					IF (status.XOPEN = 0) THEN
						StepType            := WRITE ;
					ELSE
						StepType            := OPEN ;
						Error               := TRUE;
						ErrorID             := status.XOPEN;
						Busy                := 0;
					END_IF
				WRITE:
					memset(ADR(WriteData),0,SIZEOF(WriteData));
					strcpy(ADR(WriteData),ADR('tag,0,0,#crc$R$L'));
					FrameGetBufferStruct(enable:= 1, ident:= FrameXOpenStruct.ident);
					sendbuffer				:= FrameGetBufferStruct.buffer;
					sendbufferlength		:= FrameGetBufferStruct.buflng;
					status.GetBuffer		:= FrameGetBufferStruct.status;
					IF	(status.GetBuffer = 0)	THEN
						memcpy(sendbuffer,ADR(WriteData),sendbufferlength);
						FrameWriteStruct(enable := 1, ident := FrameXOpenStruct.ident, buffer := sendbuffer,buflng := strlen(ADR(WriteData)));
						status.WRITE 				:=	FrameWriteStruct.status;
						StepType				:= READ;
					    IF (status.WRITE <> 0) THEN
							FrameReleaseOutputBufferStruct(enable:=1,ident:=FrameXOpenStruct.ident,buffer:=sendbuffer,buflng:= strlen(ADR(WriteData)));
							status.RoBuffer			:= FrameReleaseOutputBufferStruct.status;
							IF	(status.RoBuffer <> 0)	THEN
								ErrorID	:=	status.RoBuffer;
							END_IF
						END_IF
						FrameWriteStruct.enable := 0;
						FrameGetBufferStruct.enable	:= 0;
						FrameReleaseOutputBufferStruct.enable := 0;
					ELSE
						ErrorID 	:= status.GetBuffer;
						Error   	:= 1;
						Busy    	:= 0;
						StepType	:= OPEN;
						TypeOK		:= FALSE;
						FrameGetBufferStruct.enable	:= 0;
					END_IF

				READ:
					FrameReadStruct(enable:=1,ident:=FrameXOpenStruct.ident);
					ReadBuffer       	:=	FrameReadStruct.buffer;
					ReadBufferLength	:=	FrameReadStruct.buflng;
					status.READ      	:=	FrameReadStruct.status;
					IF  (status.READ = 0) THEN
						memset(ADR(ReadData),0,SIZEOF(ReadData));
						memcpy(ADR(ReadData),ReadBuffer,ReadBufferLength);                   (* copy read data into read buffer *)
						FrameReadStruct.enable	:= 0;
				        FrameReleaseBufferStruct(enable:=1, ident:=FrameXOpenStruct.ident, buffer:=ReadBuffer,buflng:=ReadBufferLength);        (* release read buffer *)
				        status.ReleaseBuffer	:=FrameReleaseBufferStruct.status;
				        IF (status.ReleaseBuffer=0) THEN
					        FrameReleaseBufferStruct.enable:=0;
							AN[0]		 :=	ReadData[0];
							AN[1]		 := ReadData[1];
							AN[2]		 := ReadData[2];
							IF	(memcmp(ADR(AN),ADR('ack'),3) = 0)	THEN
								memset(ADR(KeyType),0,SIZEOF(KeyType));
								KeyType[0] 	 :=	ReadData[6];
								KeyType[1] 	 := ReadData[7];
								KeyType[2] 	 := ReadData[8];
								KeyType[3] 	 := ReadData[9];
								IF (memcmp(ADR(KeyType),ADR('4150'),4) = 0) THEN
									StepType	:=	OPEN;
									TypeOK		:=	TRUE;
								ELSIF	(memcmp(ADR(KeyType),ADR('4102'),4) = 0) THEN
									StepType	:= 	OPEN;
									ErrorID		:=	rfidError_write_wrongType;         (*   wrong Type *)
									Error   	:=	1;
									Busy    	:=	0;
									TypeOK		:=	FALSE;
								ELSE
									StepType		:= 	OPEN;
									ErrorID			:=	rfidError_write_wrongType;            (* unknow type to write  *)
									Error   		:=	1;
									Busy    		:=	0;
									TypeOK			:=	FALSE;
								END_IF
							ELSIF	(memcmp(ADR(AN),ADR('nak'),3) = 0)	THEN
								StepType		:=	OPEN;
								ErrorID			:=	rfidError_write_failed; (* negativ answer *)
								Error   		:=	1;
								Busy    		:=	0;
								TypeOK			:=	FALSE;
							ELSE
								StepType	:= 	OPEN;
								ErrorID		:=	rfidError_write_failed; (* unknow answer *)
								Error   	:=	1;
								Busy    	:=	0;
								TypeOK			:=	FALSE;
							END_IF
						ELSE
							StepType	:=	OPEN;
							Error     	:=	1;
							ErrorID   	:=	status.ReleaseBuffer;
							Busy      	:=	0;
							TypeOK		:=	FALSE;
						END_IF
					ELSE
						memset(ADR(ReadData),0,SIZEOF(ReadData));
					END_IF
			END_CASE
		END_IF
		IF	(TypeOK	= TRUE)	THEN
			IF	(CommandReady = 0) THEN
				IF	(RegNr > 31) THEN
					Error	:=	1;
					ErrorID	:=	rfidError_write_wrongRegNr; (* hier soll ein Fehler Meldung difiniert werden: password Register, please use TP_Password Fub*)
					Busy	:=	0;
					TypeOK	:=	FALSE;
				ELSE
					itoa(RegNr,ADR(string1));
					string2:='wr,0,';
					string3:=',#crc$R$L';
					CMD	:=	strcat(ADR(string2),ADR(string1));
					CMD	:=	strcat(ADR(string2),ADR(','));
					CMD	:=	strcat(ADR(string2),Data);
					CMD	:=	strcat(ADR(string2),ADR(string3));
					memset(ADR(WriteData),0,SIZEOF(WriteData));
					strcpy(ADR(WriteData),ADR(string2));
					CommandReady:=	1;
					StepWrite	:=	WRITE;
				END_IF
			ELSE
				CASE StepWrite OF
					WRITE:
						FrameGetBufferStruct(enable:= 1, ident:= FrameXOpenStruct.ident);
						sendbuffer				:= FrameGetBufferStruct.buffer;
						sendbufferlength		:= FrameGetBufferStruct.buflng;
						status.GetBuffer		:= FrameGetBufferStruct.status;
						IF	(status.GetBuffer = 0)	THEN
							memcpy(sendbuffer,ADR(WriteData),sendbufferlength);
							FrameWriteStruct(enable := 1, ident := FrameXOpenStruct.ident, buffer := sendbuffer,buflng := strlen(ADR(WriteData)));
							status.WRITE 				:=	FrameWriteStruct.status;
						    StepWrite              		:=	READ;
						    IF (status.WRITE <> 0) THEN
								FrameReleaseOutputBufferStruct(enable:=1,ident:=FrameXOpenStruct.ident,buffer:=sendbuffer,buflng:= strlen(ADR(WriteData)));
								status.RoBuffer			:= FrameReleaseOutputBufferStruct.status;
								IF	(status.RoBuffer <> 0)	THEN
									ErrorID	:=	status.RoBuffer;
								END_IF
							END_IF
							FrameWriteStruct.enable := 0;
							FrameGetBufferStruct.enable	:= 0;
							FrameReleaseOutputBufferStruct.enable := 0;
						ELSE
							ErrorID 		:= status.GetBuffer;
							Error   		:= 1;
							Busy    		:= 0;
							StepWrite		:= WRITE;
							TypeOK			:= FALSE;
							CommandReady	:=	0;
							FrameGetBufferStruct.enable	:= 0;
						END_IF

			    	READ:
				    	FrameReadStruct(enable := 1,ident:=FrameXOpenStruct.ident);
						ReadBuffer			:=	FrameReadStruct.buffer;
						ReadBufferLength	:=	FrameReadStruct.buflng;
						status.READ			:=	FrameReadStruct.status;
						IF  (status.READ = 0)  THEN
							memset(ADR(ReadData),0,SIZEOF(ReadData));
							memcpy(ADR(ReadData),ReadBuffer,ReadBufferLength);
							FrameReadStruct.enable := 0;
					        FrameReleaseBufferStruct(enable:=1, ident:=FrameXOpenStruct.ident, buffer:=ReadBuffer,buflng:=ReadBufferLength);
					        status.ReleaseBuffer	:=	FrameReleaseBufferStruct.status;
					        IF status.ReleaseBuffer=0 THEN
								FrameReleaseBufferStruct.enable:=0;
					        	AN[0]	:= ReadData[0];
								AN[1]	:= ReadData[1];
								AN[2]	:= ReadData[2];
								IF (memcmp(ADR(AN),ADR('ack'),3) = 0) THEN
									StepWrite		:=	WRITE;
								 	Busy			:=	0;
								 	Done			:=	1;
									CommandReady	:=	0;
									TypeOK			:=	FALSE;
								ELSIF	(memcmp(ADR(AN),ADR('nak'),3) = 0)	THEN
									ERROR[0]	:=	ReadData[6];
									ERROR[1]	:=	ReadData[7];
									ERROR[2]	:=	ReadData[8];
									Error			:=	1;
									ErrorID			:=	rfidError_write_failed ;
									Busy			:=	0;
									CommandReady	:=	0;
									TypeOK			:=	FALSE;
									StepWrite		:=	WRITE;
								ELSE
									Error			:=	1;
									ErrorID			:=	rfidError_write_failed;
									Busy			:=	0;
									CommandReady	:=	0;
									TypeOK			:=	FALSE;
									StepWrite		:=	WRITE;
								END_IF
							ELSE
								Error			:=	1;
								ErrorID			:=	status.ReleaseBuffer ;
								Busy			:=	0;
								CommandReady	:=	0;
								TypeOK			:=	FALSE;
								StepWrite		:=	WRITE;
					       	END_IF
						ELSE
							memset(ADR(ReadData),0,SIZEOF(ReadData));
						END_IF
				END_CASE
			END_IF
		END_IF
	END_IF
ELSE
	Busy	:= 0;
	Error   := 0;
	ErrorID := 0;
	Done	:= 0;
END_IF
END_FUNCTION_BLOCK
```

#### TP_Read.st
```iecst
(********************************************************************
 * COPYRIGHT -- Bernecker + Rainer
 ********************************************************************
 * Library: RFID
 * File: TP_Read.st
 * Author: houx
 * Created: March 25, 2009
 *****************************************************************
;FuB: 			TP_Read
;*****************************************************************
Discription:
	This FuB is used to read the registers of the transponder.
	for this to work, the transponder must not be password-protected or a valid TP_unlock needs to be performed beforehand.
Parameter:
	Input:
		Enable(BOOL)	: The function block is only executed when enable is <> 0
		RegNr(USINT)	: Number of the register, which should be read out
	Output:
		Error(BOOL)		: Error = 0 (No Error) Error = 1(see ErrorID)
		ErrorID(BOOL)	: Number and Description in Error Table
		Busy(BOOL)		: Fub working on
		Data(BOOL)		: pointer to output Data.
		Done(BOOL)		: success, if TRUE
Author:	Xiaoguang Hou
		B&R Eggelsberg

History: 	V1.00.0 - 02 Sep 2008 first create
				V3.00.0 - 25 Mar 2009  update for serial interface transponder reader and created under AS3.0

 ********************************************************************
 * Implementation of library RFID
 ********************************************************************)

(*TODO: Add your comment here*)
FUNCTION_BLOCK TP_Read

    IF Enable = TRUE THEN
        IF ((Done = 0) AND (Error = 0)) THEN
            Busy:=TRUE;
            IF (TypeOK = FALSE) THEN
                CASE StepType OF
                    (*	------------------------------------------------	open the interface, get the internal Ident	----------------------------------------------------*)
                    OPEN:
                        FrameXOpenStruct.mode:=ADR(' /RIT=200 ');			(* long receive idle time for receive the data*)
                        FrameXOpenStruct(enable := 1,device := Ident);
                        status.XOPEN 			:= FrameXOpenStruct.status;
                        IF (status.XOPEN = 0) THEN
                            StepType            := WRITE ;
                            FrameXOpenStruct.enable := 0;
                        ELSE
                            StepType            := OPEN ;
                            Error               := TRUE;
                            ErrorID             := status.XOPEN;
                            Busy                := 0;
                            FrameXOpenStruct.enable := 0;
                        END_IF
                    WRITE:
                        memset(ADR(WriteData),0,SIZEOF(WriteData));
                        strcpy(ADR(WriteData),ADR('tag,0,#crc$R$L'));
                        FrameGetBufferStruct(enable:= 1, ident:= FrameXOpenStruct.ident);
                        sendbuffer					:= FrameGetBufferStruct.buffer;
                        sendbufferlength		:= FrameGetBufferStruct.buflng;
                        status.GetBuffer		:= FrameGetBufferStruct.status;
                        IF	(status.GetBuffer = 0)	THEN
                            memcpy(sendbuffer,ADR(WriteData),sendbufferlength);
                            FrameWriteStruct(enable := 1, ident := FrameXOpenStruct.ident, buffer := sendbuffer,buflng := strlen(ADR(WriteData)) );
                            status.WRITE 				:=	FrameWriteStruct.status;
                            IF (status.WRITE <> 0) THEN
                                FrameReleaseOutputBufferStruct(enable:=1,ident:=FrameXOpenStruct.ident,buffer:=sendbuffer,buflng:= strlen(ADR(WriteData)));
                                status.RoBuffer				:= FrameReleaseOutputBufferStruct.status;
                                IF (status.RoBuffer <> 0) THEN
                                    ErrorID:=status.RoBuffer;
                                END_IF
                            ELSE
                                StepType	:=	READ;
                                FrameWriteStruct.enable 	:= 0;
                                FrameGetBufferStruct.enable	:= 0;
                                FrameReleaseOutputBufferStruct.enable := 0;
                            END_IF
                        ELSE
                            ErrorID 	:= status.GetBuffer;
                            Error   	:= 1;
                            Busy    	:= 0;
                            StepType	:= OPEN;
                            TypeOK		:= FALSE;
                            FrameGetBufferStruct.enable	:= 0;
                        END_IF
                    READ:
                        FrameReadStruct(enable:=1,ident:=FrameXOpenStruct.ident);
                        ReadBuffer       	:=	FrameReadStruct.buffer;
                        ReadBufferLength	:=	FrameReadStruct.buflng;
                        status.READ      	:=	FrameReadStruct.status;
                        IF  (status.READ = 0) THEN
                            memset(ADR(ReadData),0,SIZEOF(ReadData));
                            memcpy(ADR(ReadData),ReadBuffer,ReadBufferLength);                   (* copy read data into read buffer *)
                            FrameReadStruct.enable	:= 0;
                            FrameReleaseBufferStruct(enable:=1, ident:=FrameXOpenStruct.ident, buffer:=ReadBuffer,buflng:=ReadBufferLength);        (* release read buffer *)
                            status.ReleaseBuffer	:=FrameReleaseBufferStruct.status;
                            IF (status.ReleaseBuffer=0) THEN
                                FrameReleaseBufferStruct.enable:=0;
                                AN[0]		 := ReadData[0];
                                AN[1]		 := ReadData[1];
                                AN[2]		 := ReadData[2];
                                IF	(memcmp(ADR(AN),ADR('ack'),3) = 0)	THEN
                                    memset(ADR(KeyType),0,SIZEOF(KeyType));
                                    KeyType[0] 	 := ReadData[6];
                                    KeyType[1] 	 := ReadData[7];
                                    KeyType[2] 	 := ReadData[8];
                                    KeyType[3] 	 := ReadData[9];
                                    IF (memcmp(ADR(KeyType),ADR('4150'),4) = 0) THEN
                                        StepType		:=	OPEN;
                                        Done         	:=	FALSE;
                                        Busy         	:=	0;
                                        CommandReady	:=	0;
                                        TypeOK			:=	TRUE;
                                    ELSIF	(memcmp(ADR(KeyType),ADR('4102'),4) = 0) THEN
                                        memset(ADR(data),0,SIZEOF(data));
                                        data[0] 	 	:=	ReadData[11];
                                        data[1] 	 	:=	ReadData[12];
                                        data[2] 	 	:=	ReadData[13];
                                        data[3] 	 	:=	ReadData[14];
                                        data[4] 	 	:=	ReadData[15];
                                        data[5] 	 	:=	ReadData[16];
                                        data[6] 	 	:=	ReadData[17];
                                        data[7] 	 	:=	ReadData[18];
                                        data[8] 	 	:=	ReadData[19];
                                        data[9] 	 	:=	ReadData[20];
                                        Data			:=	ADR(data);
                                        StepType		:=	OPEN;
                                        Done         	:=	1;
                                        Busy         	:=	0;
                                        CommandReady	:=	0;
                                        TypeOK			:=	FALSE;
                                    ELSE
                                        StepType		:= 	OPEN;
                                        ErrorID			:=	rfidError_read_wrongType;            (* wrong type to read  *)
                                        Error   		:=	1;
                                        Busy    		:=	0;
                                        CommandReady	:=	0;
                                        TypeOK			:=	FALSE;
                                    END_IF
                                ELSIF	(memcmp(ADR(AN),ADR('nak'),3) = 0)	THEN
                                    StepType		:= 	OPEN;
                                    ErrorID			:=	rfidError_read_failed; (* negativ answer *)
                                    Error   		:=	1;
                                    Busy    		:=	0;
                                    CommandReady	:=	0;
                                    TypeOK			:=	FALSE;
                                ELSE
                                    StepType		:=	OPEN;
                                    ErrorID			:=	rfidError_read_failed; (* unknow answer *)
                                    Error   		:=	1;
                                    Busy    		:=	0;
                                    CommandReady	:=	0;
                                    TypeOK			:=	FALSE;
                                END_IF
                            ELSE
                                StepType		:=	OPEN;
                                Error     		:=	1;
                                ErrorID   		:=	status.ReleaseBuffer;
                                Busy      		:=	0;
                                CommandReady	:=	0;
                                TypeOK			:=	FALSE;
                            END_IF
                        ELSE
                            memset(ADR(ReadData),0,SIZEOF(ReadData));
                        END_IF
                END_CASE
            END_IF
            IF	(TypeOK = TRUE) THEN
                IF CommandReady = 0 THEN
                    IF  ((0 < RegNr) AND (RegNr <34)) THEN
                        memset(ADR(WriteData),0,SIZEOF(WriteData));
                        CASE RegNr OF
                            REG1:
                                strcpy(ADR(WriteData),ADR('rdm,0,1,1,#crc$R$L'));
                            REG2:
                                strcpy(ADR(WriteData),ADR('rdm,0,2,1,#crc$R$L'));
                            REG3:
                                strcpy(ADR(WriteData),ADR('rdm,0,3,1,#crc$R$L'));
                            REG4:
                                strcpy(ADR(WriteData),ADR('rdm,0,4,1,#crc$R$L'));
                            REG5:
                                strcpy(ADR(WriteData),ADR('rdm,0,5,1,#crc$R$L'));
                            REG6:
                                strcpy(ADR(WriteData),ADR('rdm,0,6,1,#crc$R$L'));
                            REG7:
                                strcpy(ADR(WriteData),ADR('rdm,0,7,1,#crc$R$L'));
                            REG8:
                                strcpy(ADR(WriteData),ADR('rdm,0,8,1,#crc$R$L'));
                            REG9:
                                strcpy(ADR(WriteData),ADR('rdm,0,9,1,#crc$R$L'));
                            REG10:
                                strcpy(ADR(WriteData),ADR('rdm,0,10,1,#crc$R$L'));
                            REG11:
                                strcpy(ADR(WriteData),ADR('rdm,0,11,1,#crc$R$L'));
                            REG12:
                                strcpy(ADR(WriteData),ADR('rdm,0,12,1,#crc$R$L'));
                            REG13:
                                strcpy(ADR(WriteData),ADR('rdm,0,13,1,#crc$R$L'));
                            REG14:
                                strcpy(ADR(WriteData),ADR('rdm,0,14,1,#crc$R$L'));
                            REG15:
                                strcpy(ADR(WriteData),ADR('rdm,0,15,1,#crc$R$L'));
                            REG16:
                                strcpy(ADR(WriteData),ADR('rdm,0,16,1,#crc$R$L'));
                            REG17:
                                strcpy(ADR(WriteData),ADR('rdm,0,17,1,#crc$R$L'));
                            REG18:
                                strcpy(ADR(WriteData),ADR('rdm,0,18,1,#crc$R$L'));
                            REG19:
                                strcpy(ADR(WriteData),ADR('rdm,0,19,1,#crc$R$L'));
                            REG20:
                                strcpy(ADR(WriteData),ADR('rdm,0,20,1.#crc$R$L'));
                            REG21:
                                strcpy(ADR(WriteData),ADR('rdm,0,21,1,#crc$R$L'));
                            REG22:
                                strcpy(ADR(WriteData),ADR('rdm,0,22,1,#crc$R$L'));
                            REG23:
                                strcpy(ADR(WriteData),ADR('rdm,0,23,1,#crc$R$L'));
                            REG24:
                                strcpy(ADR(WriteData),ADR('rdm,0,24,1,#crc$R$L'));
                            REG25:
                                strcpy(ADR(WriteData),ADR('rdm,0,25,1,#crc$R$L'));
                            REG26:
                                strcpy(ADR(WriteData),ADR('rdm,0,26,1,#crc$R$L'));
                            REG27:
                                strcpy(ADR(WriteData),ADR('rdm,0,27,1,#crc$R$L'));
                            REG28:
                                strcpy(ADR(WriteData),ADR('rdm,0,28,1,#crc$R$L'));
                            REG29:
                                strcpy(ADR(WriteData),ADR('rdm,0,29,1,#crc$R$L'));
                            REG30:
                                strcpy(ADR(WriteData),ADR('rdm,0,30,1,#crc$R$L'));
                            REG31:
                                strcpy(ADR(WriteData),ADR('rdm,0,31,1,#crc$R$L'));
                            REG32:
                                strcpy(ADR(WriteData),ADR('rdm,0,32,1,#crc$R$L'));
                            REG33:
                                strcpy(ADR(WriteData),ADR('rdm,0,33,1,#crc$R$L'));
                        END_CASE
                        CommandReady:=TRUE;
                        StepREAD		:=	OPEN;
                    ELSE
                        Error   		:=	1;
                        ErrorID 		:=	rfidError_read_wrongRegNr; (* wrong register number*)
                        Busy    		:=	0;
                        CommandReady	:=	0;
                        TypeOK			:=	FALSE;
                    END_IF
                END_IF
                IF CommandReady	= 1 THEN
                    CASE StepREAD OF
                        OPEN:
                            FrameXOpenStruct.mode:=ADR('/RIT=200 ');
                            FrameXOpenStruct(enable := 1,device := Ident);
                            status.XOPEN 			:= FrameXOpenStruct.status;
                            IF (status.XOPEN = 0) THEN
                                StepREAD            := WRITE ;
                                FrameXOpenStruct.enable:=FALSE;
                            ELSE
                                StepREAD            := OPEN ;
                                Error               := TRUE;
                                ErrorID             := status.XOPEN;
                                Busy                := 0;
                                FrameXOpenStruct.enable:=FALSE;
                            END_IF
                        WRITE:
                            FrameGetBufferStruct(enable:= 1, ident:= FrameXOpenStruct.ident);
                            sendbuffer				:= FrameGetBufferStruct.buffer;
                            sendbufferlength		:= FrameGetBufferStruct.buflng;
                            status.GetBuffer		:= FrameGetBufferStruct.status;
                            IF	(status.GetBuffer = 0)	THEN
                                memcpy(sendbuffer,ADR(WriteData),SIZEOF(WriteData));
                                FrameWriteStruct(enable := 1, ident := FrameXOpenStruct.ident, buffer := sendbuffer,buflng := strlen(ADR(WriteData)));
                                status.WRITE 		:=	FrameWriteStruct.status;
                                IF (status.WRITE <> 0) THEN
                                    FrameReleaseOutputBufferStruct(enable:=1,ident:=FrameXOpenStruct.ident,buffer:=sendbuffer,buflng:= strlen(ADR(WriteData)));
                                    status.RoBuffer			:= FrameReleaseOutputBufferStruct.status;
                                    IF	(status.RoBuffer <> 0)	THEN
                                        ErrorID := status.RoBuffer;
                                        FrameReleaseOutputBufferStruct.enable:=FALSE;
                                    END_IF
                                ELSE
                                    FrameWriteStruct.enable := 0;
                                    FrameGetBufferStruct.enable	:= 0;
                                    FrameReleaseOutputBufferStruct.enable := 0;
                                    StepREAD			:=	READ;
                                END_IF
                            ELSE
                                ErrorID 		:= status.GetBuffer;
                                Error   		:= 1;
                                Busy    		:= 0;
                                StepREAD		:= OPEN;
                                TypeOK			:= FALSE;
                                CommandReady	:=	0;
                                FrameGetBufferStruct.enable	:= 0;
                            END_IF

                        READ:
                            FrameReadStruct(enable := 1,ident:=FrameXOpenStruct.ident);
                            ReadBuffer       	:=	FrameReadStruct.buffer;
                            ReadBufferLength	:=	FrameReadStruct.buflng;
                            status.READ      	:=	FrameReadStruct.status;
                            IF  (status.READ = 0)  THEN
                                memset(ADR(ReadData),0,SIZEOF(ReadData));
                                memcpy(ADR(ReadData),ReadBuffer,ReadBufferLength);
                                FrameReadStruct.enable	:=	0;
                                FrameReleaseBufferStruct(enable:=1, ident:=FrameXOpenStruct.ident, buffer:=ReadBuffer,buflng:=ReadBufferLength);
                                status.ReleaseBuffer	:=	FrameReleaseBufferStruct.status;
                                IF (status.ReleaseBuffer	= 0) THEN
                                    FrameReleaseBufferStruct.enable	:=	0;
                                    AN[0]	:= ReadData[0];
                                    AN[1]	:= ReadData[1];
                                    AN[2]	:= ReadData[2];
                                    IF (memcmp(ADR(AN),ADR('ack'),3) = 0) THEN
                                        IF ReadBufferLength <> 22 THEN
                                            StepREAD		:=	OPEN;
                                            Error       	:=	1;
                                            ErrorID      	:=	rfidError_read_failed ; (* unknow answer *)
                                            Busy         	:=	0;
                                            CommandReady	:=	0;
                                            TypeOK			:=	FALSE;
                                        ELSE
                                            StepREAD    :=	DATAREAD;
                                        END_IF
                                    ELSIF	(memcmp(ADR(AN),ADR('nak'),3) = 0)	THEN
                                        ERROR[0]	:=	ReadData[6];
                                        ERROR[1]	:=	ReadData[7];
                                        ERROR[2]	:=	ReadData[8];
                                        StepREAD		:=	OPEN;
                                        Error       	:=	1;
                                        ErrorID      	:=	atoi(ADR(ERROR)) ;
                                        Busy         	:=	0;
                                        CommandReady	:=	0;
                                        TypeOK			:=	FALSE;
                                    ELSE
                                        StepREAD		:=	OPEN;
                                        Error       	:=	1;
                                        ErrorID      	:=	rfidError_read_failed ; (* unknow answer *)
                                        Busy         	:=	0;
                                        CommandReady	:=	0;
                                        TypeOK			:=	FALSE;
                                    END_IF
                                ELSE
                                    StepREAD		:=	OPEN;
                                    Error       	:=	1;
                                    ErrorID      	:=	status.ReleaseBuffer ;
                                    Busy         	:=	0;
                                    CommandReady	:=	0;
                                    TypeOK			:=	FALSE;
                                END_IF
                            ELSE
                                memset(ADR(ReadData),0,SIZEOF(ReadData));
                            END_IF
                        DATAREAD:
                            memset(ADR(data),0,SIZEOF(data));
                            data[0] 	 	:=	ReadData[6];
                            data[1] 	 	:=	ReadData[7];
                            data[2] 	 	:=	ReadData[8];
                            data[3] 	 	:=	ReadData[9];
                            data[4] 	 	:=	ReadData[10];
                            data[5] 	 	:=	ReadData[11];
                            data[6] 	 	:=	ReadData[12];
                            data[7] 	 	:=	ReadData[13];
                            Data			:=	ADR(data);
                            Done         	:=	1;
                            Busy         	:=	0;
                            CommandReady	:=	0;
                            StepREAD     	:=	OPEN;
                            TypeOK			:=	FALSE;
                    END_CASE
                END_IF
            END_IF
        END_IF
    ELSE
        Busy:=0;
        Done:=0;
        Error:=0;
        ErrorID:=0;
        StepREAD:= 0;
        StepType:= 0;
    END_IF
END_FUNCTION_BLOCK
```

### Library Logical/Libraries/RFID_Heads (IEC)

#### RFID_Heads.fun - Exported functions and function blocks
```iecst
{REDUND_ERROR} FUNCTION_BLOCK SickHeads (*RFID hlavy SICK*) (*$GROUP=User,$CAT=User,$GROUPICON=User.png,$CATICON=User.png*)
	VAR_INPUT
		CitaciuHlavu_VYPNI : BOOL;
		PrecitajChipRFID : BOOL;
		ZapisNaChipRFID : BOOL;
		ZadaneCisloPaletky : USINT;
		Mapping_IN : ARRAY[0..7] OF USINT;
	END_VAR
	VAR_OUTPUT
		PritomnostPaletky : BOOL;
		Stav_CitaciaHlava_ON : BOOL;
		Stav_CitanieZapis_OK : BOOL;
		Stav_CitanieZapis_NG : BOOL;
		PrecitaneCisloPaletky : USINT;
		Mapping_OUT : ARRAY[0..7] OF USINT;
	END_VAR
	VAR
		Step : USINT;
		AlarmTime : TON;
	END_VAR
END_FUNCTION_BLOCK
```

#### SickHeads.st
```iecst
(* RFID hlavy SICK *)
FUNCTION_BLOCK SickHeads

	//Mapovanie//
	Stav_CitaciaHlava_ON:= Mapping_IN[0].4;
	PritomnostPaletky:= Mapping_IN[0].5;
	Mapping_OUT[0].4:= CitaciuHlavu_VYPNI;
	Mapping_OUT[1].0:= TRUE;
	Mapping_OUT[3].0:= TRUE;

	AlarmTime.PT:= T#3s;
	AlarmTime();

	CASE Step OF

		0: //Nulovanie//
			Stav_CitanieZapis_OK:= FALSE;
			Stav_CitanieZapis_NG:= FALSE;
			Mapping_OUT[0].0:= 	FALSE;
			Mapping_OUT[0].1:= 	FALSE;
			Mapping_OUT[0].2:= 	FALSE;
			Mapping_OUT[0].7:= 	FALSE;
			PrecitaneCisloPaletky:= 0;
			AlarmTime.IN:= FALSE;
			IF NOT PrecitajChipRFID AND NOT ZapisNaChipRFID THEN
				Step:= 1;
			END_IF

		1: //Čakam na kommand//
			IF PrecitajChipRFID THEN
				Step:= 10;
			ELSIF ZapisNaChipRFID THEN
				Step:= 20;
			END_IF

		10: //Čítanie//
			Mapping_OUT[0].0:= 	TRUE;
			Mapping_OUT[0].1:= 	TRUE;
			Mapping_OUT[0].2:= 	FALSE;
			Mapping_OUT[0].7:= 	TRUE;
			AlarmTime.IN:= TRUE;

			IF Mapping_IN[0].0 AND Mapping_IN[0].1 AND NOT Mapping_IN[0].2 AND Mapping_IN[0].7 THEN
				PrecitaneCisloPaletky:= Mapping_IN[4];
				Stav_CitanieZapis_OK:= TRUE;
				Step:= 11;
			ELSIF AlarmTime.Q THEN
				Stav_CitanieZapis_NG:= TRUE;
				Step:= 11;
			END_IF

		11: //Čakám na ukončenie čítania//
			IF NOT PrecitajChipRFID THEN
				Step:= 0;
			END_IF

		20: //Zápis//
			Mapping_OUT[0].0:= 	FALSE;
			Mapping_OUT[0].1:= 	FALSE;
			Mapping_OUT[0].2:= 	TRUE;
			Mapping_OUT[4]:= ZadaneCisloPaletky;
			Mapping_OUT[0].7:= 	TRUE;
			AlarmTime.IN:= TRUE;

			IF NOT Mapping_IN[0].0 AND NOT Mapping_IN[0].1 AND Mapping_IN[0].2 AND Mapping_IN[0].7 THEN
				Stav_CitanieZapis_OK:= TRUE;
				Step:= 21;
			ELSIF AlarmTime.Q THEN
				Stav_CitanieZapis_NG:= TRUE;
				Step:= 21;
			END_IF

		21: //Čakám na ukončenie zápisu//
			IF NOT ZapisNaChipRFID THEN
				Step:= 0;
			END_IF

	END_CASE

END_FUNCTION_BLOCK
```

### Library Logical/Libraries/AtlasCopco (IEC)

#### AtlasCopco.fun - Exported functions and function blocks
```iecst
{REDUND_ERROR} FUNCTION_BLOCK PrevodMomentu (*TODO: Prevod momentu s menicov atlas copco*) (*$GROUP=User,$CAT=User,$GROUPICON=User.png,$CATICON=User.png*)
	VAR_INPUT
		AtlasMaximalnaTolerancia : UDINT;
		AtlasMinimalnaTolerancia : UDINT;
		AtlasAktualnyMoment : UDINT;
	END_VAR
	VAR_OUTPUT
		ToleranciaMAX : REAL;
		ToleranciaMIN : REAL;
		AktualnyMoment : REAL;
	END_VAR
	VAR
		ByteArray2 : ARRAY[0..3] OF USINT;
		ByteArray3 : ARRAY[0..3] OF USINT;
		ByteArray1 : ARRAY[0..3] OF USINT;
		InputShifted2 : UDINT;
		InputShifted3 : UDINT;
		InputShifted1 : UDINT;
		Index2 : USINT;
		Index3 : USINT;
		Index1 : USINT;
	END_VAR
END_FUNCTION_BLOCK

{REDUND_ERROR} {REDUND_UNREPLICABLE} FUNCTION_BLOCK Round (*Zaokrúhlenie na jedno desatinné miesto*) (*$GROUP=User,$CAT=User,$GROUPICON=User.png,$CATICON=User.png*)
	VAR_INPUT
		VstupnaHodnota : {REDUND_UNREPLICABLE} UINT;
	END_VAR
	VAR_OUTPUT
		VystupnaHodnota : {REDUND_UNREPLICABLE} REAL;
	END_VAR
	VAR
		VstupnaHodnotaREAL : {REDUND_UNREPLICABLE} REAL;
		VysledokDeleniaUINT : {REDUND_UNREPLICABLE} UINT;
		VysledokDeleniaREAL : {REDUND_UNREPLICABLE} REAL;
	END_VAR
END_FUNCTION_BLOCK
```

#### PrevodMomentu.st
```iecst
(* TODO: Prevod momentu z menicov atlas copco *)
FUNCTION_BLOCK PrevodMomentu

//aktualny moment
		//rozbitie UDINT na pole USINTov
    InputShifted1:=AtlasAktualnyMoment;

    FOR Index1:=0 TO 3 DO
        ByteArray1[Index1]:=UDINT_TO_USINT(InputShifted1);
        InputShifted1:=ROR(InputShifted1,8);
    END_FOR

    //spojenie USINT do REAL vo vhodnej forme ;-)
    AktualnyMoment:=ByteArray1[3]*0.01+ByteArray1[1];

    //tolerancia MIN
    //rozbitie UDINT na pole USINTov
    InputShifted2:=AtlasMinimalnaTolerancia;

    FOR Index2:=0 TO 3 DO
        ByteArray2[Index2]:=UDINT_TO_USINT(InputShifted2);
        InputShifted2:=ROR(InputShifted2,8);
    END_FOR

    //spojenie USINT do REAL vo vhodnej forme ;-)
    ToleranciaMIN:=ByteArray2[3]*0.01+ByteArray2[1];

    //tolerancia MAX
    //rozbitie UDINT na pole USINTov
    InputShifted3:=AtlasMaximalnaTolerancia;

    FOR Index3:=0 TO 3 DO
        ByteArray3[Index3]:=UDINT_TO_USINT(InputShifted3);
        InputShifted3:=ROR(InputShifted3,8);
    END_FOR

    //spojenie USINT do REAL vo vhodnej forme ;-)
    ToleranciaMAX:=ByteArray3[3]*0.01+ByteArray3[1];
END_FUNCTION_BLOCK
```

#### Round.st - Zaokruhlenie hodnoty vysunutia srobovacky
```iecst
(* Zaokrúhlenie na jedno desatinné miesto *)
FUNCTION_BLOCK Round

    VstupnaHodnotaREAL:= UINT_TO_REAL(VstupnaHodnota);
    IF VstupnaHodnotaREAL >= 128 THEN
        VysledokDeleniaUINT:= TRUNC((VstupnaHodnotaREAL /128)*10);
        VysledokDeleniaREAL:= UINT_TO_REAL(VysledokDeleniaUINT);
        VystupnaHodnota:= VysledokDeleniaREAL /10;
    ELSE
        VystupnaHodnota:= 0;
    END_IF

END_FUNCTION_BLOCK
```

### Library Logical/Libraries/MyConvert (IEC)

#### MyConvert.fun - Exported functions and function blocks
```iecst
{REDUND_ERROR} FUNCTION_BLOCK UsintToUint (*Konvertovanie dvoch Usint do jednoho Uint*) (*$GROUP=User,$CAT=User,$GROUPICON=User.png,$CATICON=User.png*)
	VAR_INPUT
		IN_Byte0 : {REDUND_UNREPLICABLE} USINT;
		IN_Byte1 : {REDUND_UNREPLICABLE} USINT;
	END_VAR
	VAR_OUTPUT
		OUT_UINT : UINT;
	END_VAR
END_FUNCTION_BLOCK
```

#### UsintToUint.st
```iecst
(* Konvertovanie dvoch Usint do jednoho Uint *)
FUNCTION_BLOCK UsintToUint

	OUT_UINT.0:= IN_Byte0.0;
	OUT_UINT.1:= IN_Byte0.1;
	OUT_UINT.2:= IN_Byte0.2;
	OUT_UINT.3:= IN_Byte0.3;
	OUT_UINT.4:= IN_Byte0.4;
	OUT_UINT.5:= IN_Byte0.5;
	OUT_UINT.6:= IN_Byte0.6;
	OUT_UINT.7:= IN_Byte0.7;
	OUT_UINT.8:= IN_Byte1.0;
	OUT_UINT.9:= IN_Byte1.1;
	OUT_UINT.10:= IN_Byte1.2;
	OUT_UINT.11:= IN_Byte1.3;
	OUT_UINT.12:= IN_Byte1.4;
	OUT_UINT.13:= IN_Byte1.5;
	OUT_UINT.14:= IN_Byte1.6;
	OUT_UINT.15:= IN_Byte1.7;

END_FUNCTION_BLOCK
```

### Library Logical/Libraries/SkrutSety (IEC)

#### Types.typ - Exported data types
```iecst
TYPE
	PickAndPlace_CMD_typ : 	STRUCT
		ENABLE : BOOL;
		PodajSkrutku : BOOL;
		RucnyRezim : BOOL;
		RR_ZapniZasobnik : BOOL;
		RR_ZapniVibrolistu : BOOL;
		RR_OtocPodavac_Vstup : BOOL;
		RR_OtocPodavac_Vystup : BOOL;
		ResetPoruchy : BOOL;
	END_STRUCT;
	PickAndPlace_IN_typ : 	STRUCT
		ZasobnikSkrutiekPrazdny : BOOL;
		ZaplnenieListyZasobnika : BOOL;
		ZaplnenieVibrolisty_MIN : BOOL;
		ZaplnenieVibrolisty_MAX : BOOL;
		PodavacOtoceny_VSTUP : BOOL; (*Smerom k zásobníku*)
		PodavacOtoceny_VYSTUP : BOOL; (*Smerom k skrutkovačke*)
		Podavac_SkrutkaNaVstupe : BOOL;
		Podavac_SkrutkaNaVystupe : BOOL;
		NapajanieZasobnika_OK : BOOL;
		NapajanieVibrolisty_OK : BOOL;
	END_STRUCT;
	PickAndPlace_OUT_typ : 	STRUCT
		VibropohonZasobnika_RUN : BOOL;
		VibropohonListy_RUN : BOOL;
		TriediaciVzduch_RUN : BOOL; (*Tryska nad lištou zásobníka*)
		ZhadzovaciVzduch_RUN : BOOL; (*Tryska pred lištou zásobníka*)
		OtocPodavac_NaVstup : BOOL; (*Smerom k zásobníku*)
		OtocPodavac_NaVystup : BOOL; (*Smerom k skrutkovačke*)
	END_STRUCT;
	PickAndPlace_STAV_typ : 	STRUCT
		SkrutkaPripravena : BOOL;
		ERROR : BOOL;
		CisloPoruchy : USINT;
		PopisPoruchy : STRING[100];
	END_STRUCT;
	PickAndPlace_Internal_typ : 	STRUCT
		CasZaplneniaVibrolisty : TON;
		CasZaplneniaZasobnika : TON;
		CasVypnTriediacehoVzduchu : TON;
		CasPredSpustenimZasobnika : TON;
		IdleTime_200ms : TON;
		IdleTime_1s : TON;
		IdleTime_500ms : TON;
		IdleTime_100ms : TON;
		AlarmTime_10s : TON;
	END_STRUCT;
	MaticaSet_CMD_typ : 	STRUCT
		ENABLE : BOOL;
		PodajMaticu : BOOL;
		RucnyRezim : BOOL;
		RR_ZapniZasobnik : BOOL;
		RR_VysunPodavacMatic : BOOL;
		RR_OtocPodavac_Vstup : BOOL;
		RR_OtocPodavac_Vystup : BOOL;
		ResetPoruchy : BOOL;
	END_STRUCT;
	MaticaSet_IN_typ : 	STRUCT
		ZasobnikMaticPrazdny : BOOL;
		ZaplnenieListyZasobnika : BOOL;
		Oddelovac_SnimPrechoduMatice : BOOL;
		OddelovacOtoceny_VSTUP : BOOL; (*Smerom k zásobníku*)
		OddelovacOtoceny_VYSTUP : BOOL; (*Smerom k maticovačke*)
		PodavacMatice_VYSUNUTY : BOOL;
		PodavacMatice_ZASUNUTY : BOOL;
		Podavac_SnimPrechoduMatice : BOOL;
		PritomnostMaticeNaVystupe : BOOL;
		NapajanieZasobnika_OK : BOOL;
	END_STRUCT;
	MaticaSet_OUT_typ : 	STRUCT
		VibropohonZasobnika_RUN : BOOL;
		TriediaciVzduch_RUN : BOOL; (*Tryska nad lištou zásobníka*)
		ZhadzovaciVzduch_RUN : BOOL; (*Tryska pred lištou zásobníka*)
		OtocOddelovacMatice_NaVystup : BOOL; (*Smerom k maticovačke*)
		NastrelenieMatice_RUN : BOOL;
		PodavacMatice_Vysun : BOOL;
	END_STRUCT;
	MaticaSet_STAV_typ : 	STRUCT
		MaticaPripravena : BOOL;
		ERROR : BOOL;
		CisloPoruchy : USINT;
		PopisPoruchy : STRING[100];
		PodanieMatice_BUSY : BOOL;
	END_STRUCT;
	MaticaSet_Internal_typ : 	STRUCT
		PoInit : BOOL;
		CasZaplneniaZasobnika : TON;
		CasVypnTriediacehoVzduchu : TON;
		CasVypnZasobnika : TON;
		IdleTime_200ms : TON;
		IdleTime_1s : TON;
		IdleTime_500ms : TON;
		IdleTime_100ms : TON;
		AlarmTime_3s : TON;
		IdleTime_1500ms : TON;
	END_STRUCT;
END_TYPE
```

#### SkrutSety.fun - Exported functions and function blocks
```iecst
{REDUND_ERROR} FUNCTION_BLOCK PickAndPlace (*Skrutkovací set Pig and Place*) (*$GROUP=User,$CAT=User,$GROUPICON=User.png,$CATICON=User.png*)
	VAR_INPUT
		CMD : PickAndPlace_CMD_typ;
		IN : PickAndPlace_IN_typ;
	END_VAR
	VAR_OUTPUT
		OUT : PickAndPlace_OUT_typ;
		STAV : PickAndPlace_STAV_typ;
	END_VAR
	VAR
		Internal : PickAndPlace_Internal_typ;
		Step : USINT;
		zzEdge00000 : BOOL;
	END_VAR
END_FUNCTION_BLOCK

{REDUND_ERROR} FUNCTION_BLOCK MaticaSet (*Skrutkovací set maticovačky*) (*$GROUP=User,$CAT=User,$GROUPICON=User.png,$CATICON=User.png*)
	VAR_INPUT
		CMD : MaticaSet_CMD_typ;
		IN : MaticaSet_IN_typ;
	END_VAR
	VAR_OUTPUT
		OUT : MaticaSet_OUT_typ;
		STAV : MaticaSet_STAV_typ;
	END_VAR
	VAR
		Internal : MaticaSet_Internal_typ;
		Step : USINT;
	END_VAR
END_FUNCTION_BLOCK
```

#### PickAndPlace.st
```iecst
(* Skrutkovací set Pick and Place *)
FUNCTION_BLOCK PickAndPlace

	//Príznak skrutka pripravena//
	STAV.SkrutkaPripravena:= IN.Podavac_SkrutkaNaVystupe;

	//*******************************Zapnutie zásobníka keď je prázdna lišta zásobníka*****************//
	IF EDGEPOS(CMD.ENABLE = TRUE) THEN
		OUT.TriediaciVzduch_RUN:= TRUE;
		OUT.VibropohonZasobnika_RUN:= TRUE;
		OUT.VibropohonListy_RUN:= TRUE;
	END_IF

	//*******************************Ovládanie zhadzovacieho vzduchu pred lištou zásobníka******************************************//
	Internal.CasZaplneniaZasobnika.IN:= IN.ZaplnenieListyZasobnika AND OUT.VibropohonZasobnika_RUN AND IN.ZaplnenieVibrolisty_MIN AND IN.ZaplnenieVibrolisty_MAX;

	IF Internal.CasZaplneniaZasobnika.Q THEN
		OUT.ZhadzovaciVzduch_RUN:= TRUE;
	ELSE
		OUT.ZhadzovaciVzduch_RUN:= FALSE;
	END_IF

	Internal.CasZaplneniaZasobnika.PT:= T#3s;
	Internal.CasZaplneniaZasobnika();

	//******************************Vypnutie triediaceho vzduchu nad lištou zásobníka************************************************//
	Internal.CasVypnTriediacehoVzduchu.IN:= OUT.TriediaciVzduch_RUN AND NOT OUT.VibropohonZasobnika_RUN;
	IF Internal.CasVypnTriediacehoVzduchu.Q THEN
		OUT.TriediaciVzduch_RUN:= FALSE;
	END_IF

	Internal.CasVypnTriediacehoVzduchu.PT:= T#1s;
	Internal.CasVypnTriediacehoVzduchu();

	//*****************************************Vypnutie vibrolišty a zásobníka********************************************************//
	IF (OUT.VibropohonListy_RUN OR OUT.VibropohonZasobnika_RUN) AND
		IN.ZaplnenieVibrolisty_MIN AND
		IN.ZaplnenieVibrolisty_MAX AND
		IN.ZaplnenieListyZasobnika AND
		IN.PodavacOtoceny_VYSTUP AND
		NOT CMD.RR_ZapniVibrolistu AND
		NOT CMD.RR_ZapniZasobnik THEN
		Internal.CasZaplneniaVibrolisty.IN:= TRUE;
	ELSE
		Internal.CasZaplneniaVibrolisty.IN:= FALSE;
	END_IF

	IF (OUT.VibropohonListy_RUN OR OUT.VibropohonZasobnika_RUN) AND Internal.CasZaplneniaVibrolisty.Q THEN
		OUT.VibropohonListy_RUN:= FALSE;
		OUT.VibropohonZasobnika_RUN:= FALSE;
	END_IF

	Internal.CasZaplneniaVibrolisty.PT:= T#2s;
	Internal.CasZaplneniaVibrolisty();

	//***********************************Enable knižnice***************************************//
	IF NOT CMD.ENABLE AND Step <> 0 THEN
		OUT.VibropohonListy_RUN:= FALSE;
		OUT.VibropohonZasobnika_RUN:= FALSE;
		OUT.ZhadzovaciVzduch_RUN:= FALSE;
		Step:= 0;
	END_IF

	//**********************************Reset poruchy*****************************************//
	//1 - porucha otočenia podavača smerom k zasobniku
	//2 - porucha otočenia podavača smerom k skrutkovačke
	//3 - porucha snímača skrutky na vystupe podavača

	IF CMD.ResetPoruchy OR NOT CMD.ENABLE THEN
		STAV.ERROR:= FALSE;
		STAV.CisloPoruchy:= 0;
		STAV.PopisPoruchy:= '';
	END_IF

	CASE Step OF

		0: //Nulovanie//
			Internal.IdleTime_200ms.IN:= FALSE;
			Internal.IdleTime_100ms.IN:= FALSE;
			Internal.IdleTime_500ms.IN:= FALSE;
			Internal.IdleTime_1s.IN:= FALSE;
			Internal.AlarmTime_10s.IN:= FALSE;
			CMD.PodajSkrutku:= FALSE;
			CMD.RR_ZapniVibrolistu:= FALSE;
			CMD.RR_ZapniZasobnik:= FALSE;
			CMD.RR_OtocPodavac_Vstup:= FALSE;
			CMD.RR_OtocPodavac_Vystup:= FALSE;
			CMD.RucnyRezim:= FALSE;
			IF NOT CMD.PodajSkrutku AND CMD.ENABLE AND NOT STAV.ERROR THEN
				Step:= 1;
			END_IF

		1: //Čakam na spustenie//
			Internal.IdleTime_1s.IN:= NOT IN.Podavac_SkrutkaNaVystupe;

			IF Internal.IdleTime_1s.Q THEN
				CMD.PodajSkrutku:= TRUE;
			END_IF

			IF CMD.RucnyRezim THEN
				Step:= 70;
			ELSIF CMD.PodajSkrutku THEN
				Internal.IdleTime_1s.IN:= FALSE;
				Step:= 10;
			END_IF

		10: //Kontrola skrutky na vystupe podavaca//
			IF IN.Podavac_SkrutkaNaVystupe THEN
				Step:= 0;
			ELSE
				Step:= 11;
			END_IF

		11: //Otocenie podavaca na vstup smerom k zasobniku//
			OUT.OtocPodavac_NaVystup:= FALSE;
			OUT.OtocPodavac_NaVstup:= TRUE;
			Internal.AlarmTime_10s.IN:= TRUE;

			Internal.IdleTime_1s.IN:= IN.PodavacOtoceny_VSTUP;

			IF Internal.IdleTime_1s.Q THEN
				Internal.AlarmTime_10s.IN:= FALSE;
				Internal.IdleTime_1s.IN:= FALSE;
				Step:= 15;
			ELSIF Internal.AlarmTime_10s.Q THEN
				STAV.ERROR:= TRUE;
				STAV.CisloPoruchy:= 1;
				STAV.PopisPoruchy:= 'Porucha snimaca otocenia podavaca na vstup';
				Step:= 0;
			END_IF

		15: //Kontrola zaplnenie vibrolisty//
			IF IN.ZaplnenieVibrolisty_MAX AND IN.ZaplnenieVibrolisty_MIN AND IN.ZaplnenieListyZasobnika THEN
				Internal.IdleTime_500ms.IN:= FALSE;
				Step:= 20;
			ELSE
				Internal.IdleTime_1s.IN:= FALSE;
				Internal.IdleTime_200ms.IN:= FALSE;
				Step:= 30;
			END_IF

		20: //Spustenie vibrolisty//
			OUT.VibropohonListy_RUN:= TRUE;
			Internal.IdleTime_500ms.IN:= IN.Podavac_SkrutkaNaVstupe;

			IF Internal.IdleTime_500ms.Q THEN
				Internal.IdleTime_500ms.IN:= FALSE;
				Step:= 21;
			END_IF

		21: //Otocenie podavaca na vystup smerom k skrutkovacke//
			OUT.OtocPodavac_NaVstup:= FALSE;
			OUT.OtocPodavac_NaVystup:= TRUE;

			Internal.AlarmTime_10s.IN:= NOT IN.PodavacOtoceny_VYSTUP;

			Internal.IdleTime_1s.IN:= IN.PodavacOtoceny_VYSTUP;

			IF Internal.IdleTime_1s.Q AND IN.Podavac_SkrutkaNaVystupe THEN
				OUT.VibropohonListy_RUN:= FALSE;
				Step:= 0;
			ELSIF Internal.IdleTime_1s.Q AND NOT IN.Podavac_SkrutkaNaVystupe THEN
				Internal.IdleTime_1s.IN:= FALSE;
				Internal.AlarmTime_10s.IN:= FALSE;
				Step:= 11;
			ELSIF Internal.AlarmTime_10s.Q THEN
				STAV.ERROR:= TRUE;
				STAV.CisloPoruchy:= 2;
				STAV.PopisPoruchy:= 'Porucha snimaca otocenia podavaca na vystup';
				Step:= 0;
			END_IF

		30: //Spustenie vibrolisty a zasobnika//
			OUT.TriediaciVzduch_RUN:= TRUE;
			OUT.VibropohonListy_RUN:= TRUE;

			Internal.IdleTime_1s.IN:= OUT.TriediaciVzduch_RUN;
			Internal.IdleTime_200ms.IN:= IN.Podavac_SkrutkaNaVstupe AND OUT.VibropohonZasobnika_RUN;

			IF Internal.IdleTime_1s.Q THEN
				OUT.VibropohonZasobnika_RUN:= TRUE;
			END_IF

			IF Internal.IdleTime_200ms.Q THEN
				Internal.IdleTime_1s.IN:= FALSE;
				Internal.IdleTime_200ms.IN:= FALSE;
				Step:= 31;
			END_IF

		31: //Otocenie podavaca na vystup smerom k skrutkovacke//
			OUT.OtocPodavac_NaVstup:= FALSE;
			OUT.OtocPodavac_NaVystup:= TRUE;

			Internal.AlarmTime_10s.IN:= NOT IN.PodavacOtoceny_VYSTUP;

			Internal.IdleTime_1s.IN:= IN.PodavacOtoceny_VYSTUP;

			IF Internal.IdleTime_1s.Q AND IN.Podavac_SkrutkaNaVystupe THEN
				Internal.IdleTime_1s.IN:= FALSE;
				Step:= 0;
			ELSIF Internal.IdleTime_1s.Q AND NOT IN.Podavac_SkrutkaNaVystupe THEN
				Internal.IdleTime_1s.IN:= FALSE;
				Internal.AlarmTime_10s.IN:= FALSE;
				Step:= 11;
			ELSIF Internal.AlarmTime_10s.Q THEN
				STAV.ERROR:= TRUE;
				STAV.CisloPoruchy:= 2;
				STAV.PopisPoruchy:= 'Porucha snimaca otocenia podavaca na vystup';
				Step:= 0;
			END_IF

		70: //Rucny rezim//
			OUT.VibropohonListy_RUN:= CMD.RR_ZapniVibrolistu;

			IF CMD.RR_ZapniZasobnik THEN
				OUT.TriediaciVzduch_RUN:= TRUE;
				Internal.IdleTime_1s.IN:= TRUE;
			ELSE
				Internal.IdleTime_1s.IN:= FALSE;
			END_IF

			OUT.VibropohonZasobnika_RUN:= Internal.IdleTime_1s.Q;

			IF NOT CMD.RucnyRezim THEN
				OUT.VibropohonListy_RUN:= FALSE;
				OUT.VibropohonZasobnika_RUN:= FALSE;
				Step:= 0;
			ELSIF CMD.PodajSkrutku THEN
				Step:= 10;
			END_IF

			IF CMD.RR_OtocPodavac_Vstup THEN
				OUT.OtocPodavac_NaVystup:= FALSE;
				OUT.OtocPodavac_NaVstup:= TRUE;
				CMD.RR_OtocPodavac_Vstup:= FALSE;
			ELSIF CMD.RR_OtocPodavac_Vystup THEN
				OUT.OtocPodavac_NaVstup:= FALSE;
				OUT.OtocPodavac_NaVystup:= TRUE;
				CMD.RR_OtocPodavac_Vystup:= FALSE;
			END_IF

	END_CASE

	//*****************Časovače************************//
	Internal.IdleTime_100ms.PT:= T#200ms;
	Internal.IdleTime_100ms();
	Internal.IdleTime_200ms.PT:= T#200ms;
	Internal.IdleTime_200ms();
	Internal.IdleTime_500ms.PT:= T#200ms;
	Internal.IdleTime_500ms();
	Internal.IdleTime_1s.PT:= T#1s;
	Internal.IdleTime_1s();
	Internal.AlarmTime_10s.PT:= T#10s;
	Internal.AlarmTime_10s();
	Internal.CasPredSpustenimZasobnika.PT:= T#1s;
	Internal.CasPredSpustenimZasobnika();

END_FUNCTION_BLOCK
```
